(* CODESYS project string-builder.library
   Description: The standard ``CONCAT`` function is really cumbersome to use to build complex
      strings. This library implements a string builder method and some string format
      functions.
   Author: John te Bokkel
   Version: 0.5.0.0
   Company: PowerCore Engineering
   Title: StringBuilder32
   Placeholder: StringBuilder
   LanguageModelAttribute: qualified-access-only
   DefaultNamespace: PSB
   DocFormat: reStructuredText

Project tree, tasks and I/O mapping:
  libraries: CAA Types Extern, 3.5.17.0 (CAA Technical Workgroup); CAA FB Factory, 3.5.17.0 (CAA Technical Workgroup); Common Behaviour Model, 3.5.17.0 (3S - Smart Software Solutions GmbH); StringUtils, 3.5.18.0 (System); StringBuilder Interfaces32, * (PowerCore Engineering); MemoryUtils, * (3S - Smart Software Solutions GmbH)
  StringBuilder/
    Enums/
      data type Alignment
      data type ERROR
    Functions/
      function Align_String [ST]
      function ANY_TO_NUMSTRING [ST]
      function AppendStringNTimes [ST]
      function DIGIT_TO_CHAR [ST]
      FormatExt/
        function FormatExt_10 [ST]
        function FormatExt_1 [ST]
        function FormatExt_2 [ST]
        function FormatExt_3 [ST]
        function FormatExt_4 [ST]
        function FormatExt_5 [ST]
        function FormatExt_6 [ST]
        function FormatExt_7 [ST]
        function FormatExt_8 [ST]
        function FormatExt_9 [ST]
        function FormatExt_ArrayOfStr [ST]
      function Format_10 [ST]
      function Format_1 [ST]
      function Format_2 [ST]
      function Format_3 [ST]
      function Format_4 [ST]
      function Format_5 [ST]
      function Format_6 [ST]
      function Format_7 [ST]
      function Format_8 [ST]
      function Format_9 [ST]
      function Format_ArrayOfStr [ST]
      function POINTER_TO_STRING [ST]
    Function Blocks/
      function block StringBuilderExt [ST]: Append, p_CharBufferPtr, p_length, Reset
      function block StringBuilder [ST]: Append, p_CharBufferPtr, p_length, Reset
    GlobalConstants/
      global variables Constants
    GlobalVariables/
      global variables Variables
    Interfaces/
    Internal/
      function FindFormat [ST]
    Structs/
      data type FormatOptions
      data type slice
    Templates/
      Behaviour Model/
        function block ETrigATlTo_Temp [ST]: CleanupAction, CyclicAction, ExitAction, ResetAction, SampleAction, StartAction
        function block ETrigATl_Temp [ST]: CleanupAction, CyclicAction, ExitAction, ResetAction, SampleAction, StartAction
        function block ETrigATo_Temp [ST]: CleanupAction, CyclicAction, ExitAction, ResetAction, SampleAction, StartAction
        function block ETrigA_Temp [ST]: CleanupAction, CyclicAction, ExitAction, ResetAction, SampleAction, StartAction
        function block ETrigTlTo_Temp [ST]: CleanupAction, CyclicAction, ExitAction, ResetAction, SampleAction, StartAction
        function block ETrigTl_Temp [ST]: CleanupAction, CyclicAction, ExitAction, ResetAction, SampleAction, StartAction
        function block ETrigTo_Temp [ST]: CleanupAction, CyclicAction, ExitAction, ResetAction, SampleAction, StartAction
        function block ETrig_Temp [ST]: CleanupAction, CyclicAction, ExitAction, ResetAction, SampleAction, StartAction
        function block LConC_Temp [ST]: CleanupAction, CyclicAction, ExitAction, ResetAction, StartAction
        function block LConTlC_Temp [ST]: CleanupAction, CyclicAction, ExitAction, ResetAction, StartAction
        function block LConTlTo_Temp [ST]: CleanupAction, CyclicAction, ExitAction, ResetAction, StartAction
        function block LConTl_Temp [ST]: CleanupAction, CyclicAction, ExitAction, ResetAction, StartAction
        function block LConTo_Temp [ST]: CleanupAction, CyclicAction, ExitAction, ResetAction, StartAction
        function block LCon_Temp [ST]: CleanupAction, CyclicAction, ExitAction, ResetAction, StartAction
      FB Factory/
        function block CustomData [ST]
        function block CustomFBFactory_heap [ST]: Create, prvInstCount, prvInstPoolExtendsFactor, prvInstSize
        function block CustomFBFactory_static [ST]: Create, prvInstPoolAdr, prvInstPoolSize, prvInstSize
        function block CustomFB [ST]: prvInstInit
    Types/
*)

// StringBuilder/Enums/Alignment
{attribute 'qualified_only'}
{attribute 'strict'}
TYPE Alignment :
(
	Left,
	Center,
	Right
);
END_TYPE

// StringBuilder/Enums/ERROR
{attribute 'qualified_only'}
//{attribute 'conditionalshow'}
//{attribute 'conditionalshow' := 'SomeText'}
//{attribute 'hide'}
TYPE ERROR : (NO_ERROR, TIME_OUT); END_TYPE

// StringBuilder/Structs/FormatOptions
TYPE FormatOptions :
STRUCT
	// how many decimals a formatted number should have
	iPrecision : INT := -1;
	// the min width of the field in characters (if less than 0 no padding or alignment is performed)
	iMinWidth : INT := -1;
	// how the text is aligned
	align : Alignment := Alignment.Right;
	// A single character which is used to pad the formatted text
	sFill : STRING(1) := ' '; 
END_STRUCT
END_TYPE

// StringBuilder/Structs/slice
TYPE slice :
STRUCT
	start : DINT;
	end : DINT;
END_STRUCT
END_TYPE

// StringBuilder/GlobalConstants/Constants
{attribute 'qualified_only'}
VAR_GLOBAL CONSTANT
	gc_fmtPointerOptions : FormatOptions := (iMinWidth:=16, align:=Alignment.Right, sFill:='0');
END_VAR

// StringBuilder/GlobalVariables/Variables
{attribute 'qualified_only'}
//{attribute 'conditionalshow'}
//{attribute 'conditionalshow' := 'SomeText'}
//{attribute 'hide'}
VAR_GLOBAL
	g_iDummy : INT; /// This is a dummy global variable
END_VAR

// StringBuilder/Functions/Align_String
FUNCTION Align_String : BOOL
VAR_INPUT
	itfStringBuilder : PSBItfs.IStringBuilder;
	sVal : STRING(255);
	options : FormatOptions;
END_VAR
VAR
	iWidth : INT;
	iPadding : INT;
	iLeft : INT;
	iRight : INT;
END_VAR

Align_String := TRUE;
IF itfStringBuilder <> 0 THEN
	IF options.iMinWidth >= 0 THEN
		iWidth := DINT_TO_INT(Stu.StrLenA(ADR(sVal)));
		IF iWidth < options.iMinWidth THEN
			iPadding := options.iMinWidth - iWidth;
		ELSE
			iPadding := 0;
		END_IF
		
		IF iPadding = 0 THEN
			itfStringBuilder.Append(sVal);
			RETURN;
		END_IF
		
		CASE options.align OF
			Alignment.Left:
				itfStringBuilder.Append(sVal);
				AppendStringNTimes(itfStringBuilder, options.sFill, iPadding);
			Alignment.Center:
				iLeft := iPadding / 2;
				iRight := (iPadding + 1) / 2;
				AppendStringNTimes(itfStringBuilder, options.sFill, iLeft);
				itfStringBuilder.Append(sVal);
				AppendStringNTimes(itfStringBuilder, options.sFill, iRight);
			Alignment.Right:
				AppendStringNTimes(itfStringBuilder, options.sFill, iPadding);
				itfStringBuilder.Append(sVal);
		END_CASE
	ELSE
		itfStringBuilder.Append(sVal);
	END_IF
ELSE
	Align_String := FALSE;
END_IF

END_FUNCTION

// StringBuilder/Functions/AppendStringNTimes
FUNCTION AppendStringNTimes : BOOL
VAR_INPUT
	itfStringBuilder : PSBItfs.IStringBuilder;
	sVal : STRING(1);
	iTimes : INT;
END_VAR
VAR
	ix : INT;
END_VAR

AppendStringNTimes := TRUE;
IF itfStringBuilder <> 0 THEN
	IF iTimes > 0 THEN
		FOR ix:=0 TO (iTimes - 1) BY 1 DO
			itfStringBuilder.Append(sVal);
		END_FOR
	END_IF
ELSE
	AppendStringNTimes := FALSE;
END_IF

END_FUNCTION

// StringBuilder/Functions/ANY_TO_NUMSTRING
FUNCTION ANY_TO_NUMSTRING : STRING(129)
VAR_INPUT
	in : ANY;
	base : BYTE;
	xLoCase : BOOL;
	options : FormatOptions;
END_VAR
VAR
	sb : StringBuilder;
	pResult : POINTER TO STRING(129);
	aBuf : ARRAY [0..129] OF BYTE;
	value : UDINT;
	wValue : WORD;
	dwValue : DWORD;
	siValue : SINT;
	iValue : INT;
	diValue : DINT;
	liValue : LINT;
	xSigned : BOOL;
	digit : BYTE;
	ix : BYTE;
	_base : UDINT;
END_VAR

CASE in.TypeClass OF
	__SYSTEM.TYPE_CLASS.TYPE_BOOL:
		value := BYTE_TO_UDINT(in.pValue^);
	__SYSTEM.TYPE_CLASS.TYPE_BIT:
		value := BYTE_TO_UDINT(in.pValue^);
	__SYSTEM.TYPE_CLASS.TYPE_BYTE:
		value := BYTE_TO_UDINT(in.pValue^);
	__SYSTEM.TYPE_CLASS.TYPE_WORD:
		MEMUtils.MemCpy(ADR(wValue), in.pValue, SIZEOF(WORD));
		value := WORD_TO_UDINT(wValue);
	__SYSTEM.TYPE_CLASS.TYPE_DWORD:
		MEMUtils.MemCpy(ADR(dwValue), in.pValue, SIZEOF(DWORD));
		value := DWORD_TO_UDINT(dwValue);
	__SYSTEM.TYPE_CLASS.TYPE_LWORD:
		MEMUtils.MemCpy(ADR(value), in.pValue, SIZEOF(LWORD));
	__SYSTEM.TYPE_CLASS.TYPE_SINT:
		MEMUtils.MemCpy(ADR(siValue), in.pValue, SIZEOF(SINT));
		xSigned := siValue < 0;
		value := SINT_TO_UDINT(ABS(siValue));
	__SYSTEM.TYPE_CLASS.TYPE_INT:
		MEMUtils.MemCpy(ADR(iValue), in.pValue, SIZEOF(INT));
		xSigned := iValue < 0;
		value := INT_TO_UDINT(ABS(iValue));
	__SYSTEM.TYPE_CLASS.TYPE_DINT:
		MEMUtils.MemCpy(ADR(diValue), in.pValue, SIZEOF(DINT));
		xSigned := diValue < 0;
		value := DINT_TO_UDINT(ABS(diValue));
	__SYSTEM.TYPE_CLASS.TYPE_LINT:
		MEMUtils.MemCpy(ADR(liValue), in.pValue, SIZEOF(LINT));
		xSigned := liValue < 0;
		value := LINT_TO_UDINT(ABS(liValue));
	__SYSTEM.TYPE_CLASS.TYPE_USINT:
		value := BYTE_TO_UDINT(in.pValue^);
	__SYSTEM.TYPE_CLASS.TYPE_UINT:
		MEMUtils.MemCpy(ADR(wValue), in.pValue, SIZEOF(UINT));
		value := WORD_TO_UDINT(wValue);
	__SYSTEM.TYPE_CLASS.TYPE_UDINT:
		MEMUtils.MemCpy(ADR(dwValue), in.pValue, SIZEOF(UDINT));
		value := DWORD_TO_UDINT(dwValue);
	__SYSTEM.TYPE_CLASS.TYPE_ULINT:
		MEMUtils.MemCpy(ADR(value), in.pValue, SIZEOF(ULINT));
	__SYSTEM.TYPE_CLASS.TYPE_REAL:
		MEMUtils.MemCpy(ADR(dwValue), in.pValue, SIZEOF(REAL));
		value := DWORD_TO_UDINT(dwValue);
	__SYSTEM.TYPE_CLASS.TYPE_LREAL:
		MEMUtils.MemCpy(ADR(value), in.pValue, SIZEOF(LREAL));
	(* __SYSTEM.TYPE_CLASS.TYPE_STRING:
	__SYSTEM.TYPE_CLASS.TYPE_WSTRING: *)
	__SYSTEM.TYPE_CLASS.TYPE_TIME:
		MEMUtils.MemCpy(ADR(dwValue), in.pValue, SIZEOF(TIME));
		value := DWORD_TO_UDINT(dwValue);
	__SYSTEM.TYPE_CLASS.TYPE_DATE:
		MEMUtils.MemCpy(ADR(dwValue), in.pValue, SIZEOF(DATE));
		value := DWORD_TO_UDINT(dwValue);
	__SYSTEM.TYPE_CLASS.TYPE_DATEANDTIME:
		MEMUtils.MemCpy(ADR(dwValue), in.pValue, SIZEOF(DT));
		value := DWORD_TO_UDINT(dwValue);
	__SYSTEM.TYPE_CLASS.TYPE_TIMEOFDAY:
		MEMUtils.MemCpy(ADR(dwValue), in.pValue, SIZEOF(TOD));
		value := DWORD_TO_UDINT(dwValue);
	(*__SYSTEM.TYPE_CLASS.TYPE_POINTER:
	__SYSTEM.TYPE_CLASS.TYPE_REFERENCE:
	__SYSTEM.TYPE_CLASS.TYPE_SUBRANGE:
	__SYSTEM.TYPE_CLASS.TYPE_ENUM:
	__SYSTEM.TYPE_CLASS.TYPE_ARRAY:
	__SYSTEM.TYPE_CLASS.TYPE_PARAMS:
	__SYSTEM.TYPE_CLASS.TYPE_USERDEF:
	__SYSTEM.TYPE_CLASS.TYPE_NONE:
	__SYSTEM.TYPE_CLASS.TYPE_ANY:
	__SYSTEM.TYPE_CLASS.TYPE_ANYBIT:
	__SYSTEM.TYPE_CLASS.TYPE_ANYDATE:
	__SYSTEM.TYPE_CLASS.TYPE_ANYINT:
	__SYSTEM.TYPE_CLASS.TYPE_ANYNUM:
	__SYSTEM.TYPE_CLASS.TYPE_ANYREAL:
	__SYSTEM.TYPE_CLASS.TYPE_LAZY: *)
	__SYSTEM.TYPE_CLASS.TYPE_LTIME:
		MEMUtils.MemCpy(ADR(value), in.pValue, SIZEOF(LTIME));
	__SYSTEM.TYPE_CLASS.TYPE_LDATE:
		MEMUtils.MemCpy(ADR(value), in.pValue, SIZEOF(LDATE));
	__SYSTEM.TYPE_CLASS.TYPE_LDATEANDTIME:
		MEMUtils.MemCpy(ADR(value), in.pValue, SIZEOF(LDT));
	(*__SYSTEM.TYPE_CLASS.TYPE_BITCONST: *)
	ELSE
		// Anything not explicitly handled will return the pointer value
		value := __XWORD_TO_UDINT(in.pValue);
END_CASE

ix := 129;
_base := BYTE_TO_UDINT(base);
WHILE TRUE DO
	digit := UDINT_TO_BYTE(value MOD _base);
	ix := ix - 1;
	aBuf[ix] := DIGIT_TO_CHAR(digit, xLoCase);
	value := value / _base;
	IF value = 0 OR (xSigned AND ix = 1) OR (NOT xSigned AND ix = 0) THEN
		EXIT;
	END_IF
END_WHILE

IF xSigned THEN
	ix := ix - 1;
	aBuf[ix] := 45; // '-'
END_IF

pResult := ADR(aBuf[ix]);

Align_String(sb, pResult^, options);
ANY_TO_NUMSTRING := sb.sOutput;

END_FUNCTION

// StringBuilder/Functions/DIGIT_TO_CHAR
FUNCTION DIGIT_TO_CHAR : BYTE
VAR_INPUT
	digit : BYTE;
	xLoCase : BOOL;
END_VAR
VAR
END_VAR

IF digit < 10 THEN
	DIGIT_TO_CHAR := digit + 48; // '0' = 48
ELSE
	IF xLoCase THEN
		DIGIT_TO_CHAR := digit + 97 - 10; // 'a' = 97
	ELSE
		DIGIT_TO_CHAR := digit + 65 - 10; // 'A' = 65
	END_IF	
END_IF

END_FUNCTION

// StringBuilder/Function Blocks/StringBuilder
{attribute 'analysis' := '-2'} // empty function block
FUNCTION_BLOCK StringBuilder IMPLEMENTS PSBItfs.IStringBuilder
VAR_INPUT
END_VAR
VAR_OUTPUT
	sOutput : STRING(255);
END_VAR
VAR
	ix : DINT;
END_VAR

METHOD PUBLIC Append : INT
VAR_INPUT
	sVal : STRING(255);
END_VAR
VAR
	diCpy : DINT;
	diCpyInter : DINT;
END_VAR
IF ix = 0 THEN
	sOutput := sVal;
	ix := MAX(Stu.StrLenA(ADR(sOutput)), 0);
	Append := DINT_TO_INT(ix);
ELSIF ix >= 255 THEN
	Append := 0;
ELSE
	
	diCpyInter := Stu.StrCpyA(ADR(sOutput[ix]), MAX(0, 255-ix), ADR(sVal));
	// Working around TM258 PLC StrCpyA not actually returning the number of copied characters
	IF diCpyInter = 0 THEN
		// need to add one for the \0 that StrCpyA should count
		diCpyInter := MIN(Stu.StrLenA(ADR(sVal)) + 1, 255-ix);
	END_IF
	// 1 less than StrCpyA because that value includes \0 (NULL) terminator
	diCpy := MAX(diCpyInter - 1, 0);
	
	Append := DINT_TO_INT(diCpy);
	ix := ix + diCpy;
	// ensure we always have null termination
	sOutput[ix+1] := 0;
END_IF
END_METHOD

PROPERTY p_CharBufferPtr : POINTER TO BYTE
GET
p_CharBufferPtr := ADR(sOutput);
END_GET
END_PROPERTY

PROPERTY p_length : UDINT
GET
p_length := DINT_TO_UDINT(ix);
END_GET
END_PROPERTY

METHOD Reset : BOOL
VAR_INPUT
END_VAR
sOutput := '';
ix := 0;
END_METHOD

END_FUNCTION_BLOCK

// StringBuilder/Functions/Format_10
/// String format ``fmtstr`` with values in ``str1``, etc.
FUNCTION Format_10 : STRING(255)
VAR_INPUT
	fmtstr : STRING(255);
	str1 : STRING(255);
	str2 : STRING(255);
	str3 : STRING(255);
	str4 : STRING(255);
	str5 : STRING(255);
	str6 : STRING(255);
	str7 : STRING(255);
	str8 : STRING(255);
	str9 : STRING(255);
	str10 : STRING(255);
END_VAR
VAR
	apStr : ARRAY [0..9] OF POINTER TO STRING(255) := [ADR(str1), ADR(str2), ADR(str3), ADR(str4), ADR(str5),
	                                                   ADR(str6), ADR(str7), ADR(str8), ADR(str9), ADR(str10)];
END_VAR

Format_10 := Format_ArrayOfStr(fmtstr, ADR(apStr), 10);

END_FUNCTION

// StringBuilder/Functions/Format_ArrayOfStr
/// Replace ``uiElements`` number of ``{}`` with the sequential values in array. 
FUNCTION Format_ArrayOfStr : STRING(255)
VAR_INPUT
	fmtstr : STRING(255);
	// pArray is cast to: POINTER TO ARRAY [0..99] OF POINTER TO STRING(255);
	pArray : POINTER TO BYTE;
	// Actual number of elements in array
	uiElements : UINT;
END_VAR
VAR
	papStr : POINTER TO ARRAY [0..99] OF POINTER TO STRING(255);
	ix : UINT;
	sb : StringBuilder;
	fmtAt : slice;
	last : slice;
	substr : STRING(255);
	iLenRemaining : INT;
	iPos : INT;
END_VAR

papStr := pArray;
fmtAt := FindFormat(fmtstr, 1);

IF fmtAt.start <= 0 THEN
	Format_ArrayOfStr := fmtstr;
	// no format strings found so just return
	RETURN;
END_IF

last.end := 1;
iPos:=1;

FOR ix:=0 TO MIN((uiElements - 1), 99) BY 1 DO
	Stu.StrMidA(pst:=ADR(fmtstr),
				uiInputBufferSize:=SIZEOF(fmtstr),
				iLength:=DINT_TO_INT(fmtAt.start) - iPos,
				iPosition:=iPos,
				pstResult:=ADR(substr),
				uiResultBufferSize:=SIZEOF(substr));
	sb.Append(substr);
	sb.Append(papStr^[ix]^);
	last := fmtAt;
	iPos := DINT_TO_INT(last.end+1);
	fmtAt := FindFormat(fmtstr, fmtAt.end);
	IF fmtAt.start <= 0 THEN
		EXIT;
	END_IF
END_FOR

iLenRemaining := DINT_TO_INT(Stu.StrLenA(ADR(fmtstr[last.end])));
IF iLenRemaining > 0 THEN
	Stu.StrMidA(pst:=ADR(fmtstr),
				uiInputBufferSize:=SIZEOF(fmtstr),
				iLength:=iLenRemaining,
				iPosition:=DINT_TO_INT(last.end+1),
				pstResult:=ADR(substr),
				uiResultBufferSize:=SIZEOF(substr));
	sb.Append(substr);
END_IF
Format_ArrayOfStr := sb.sOutput;

END_FUNCTION

// StringBuilder/Internal/FindFormat
/// Find the format string
{attribute 'conditionalshow' := 'Developer'}
FUNCTION FindFormat : slice
VAR_IN_OUT CONSTANT
	fmtstr : STRING(255);
END_VAR
VAR_INPUT
	start : DINT;
END_VAR
VAR
END_VAR
VAR CONSTANT
	FMT : STRING(2) := '{}';
END_VAR

// lets start out with really basic
// this could evolve into a lexer based system with format directives 
// etc, but lets just start with what we need today.

FindFormat.start := Stu.StrFindA(ADR(fmtstr), ADR(FMT), DINT_TO_UINT(start));
IF FindFormat.start > 0 THEN
	FindFormat.end := FindFormat.start + 1;
END_IF

END_FUNCTION

// StringBuilder/Functions/Format_1
/// String format ``fmtstr`` with values in ``str1``, etc.
FUNCTION Format_1 : STRING(255)
VAR_INPUT
	fmtstr : STRING(255);
	str1 : STRING(255);
END_VAR
VAR
	sb : StringBuilder;
	fmtAt : slice;
	substr : STRING(255);
	iLenRemaining : INT;
END_VAR

fmtAt := FindFormat(fmtstr, 1);
IF fmtAt.start <= 0 THEN
	Format_1 := fmtstr;
ELSE
	Stu.StrMidA(pst:=ADR(fmtstr), uiInputBufferSize:=SIZEOF(fmtstr), iLength:=DINT_TO_INT(fmtAt.start - 1), iPosition:=1, pstResult:=ADR(substr), uiResultBufferSize:=SIZEOF(substr));
	sb.Append(substr);
	sb.Append(str1);
	iLenRemaining := DINT_TO_INT(Stu.StrLenA(ADR(fmtstr[fmtAt.end])));
	IF iLenRemaining > 0 THEN
		Stu.StrMidA(pst:=ADR(fmtstr), uiInputBufferSize:=SIZEOF(fmtstr), iLength:=iLenRemaining, iPosition:=DINT_TO_INT(fmtAt.end+1), pstResult:=ADR(substr), uiResultBufferSize:=SIZEOF(substr));
		sb.Append(substr);
	END_IF
	Format_1 := sb.sOutput;
END_IF

END_FUNCTION

// StringBuilder/Functions/Format_2
/// String format ``fmtstr`` with values in ``str1``, etc.
FUNCTION Format_2 : STRING(255)
VAR_INPUT
	fmtstr : STRING(255);
	str1 : STRING(255);
	str2 : STRING(255);
END_VAR
VAR
	apStr : ARRAY [0..1] OF POINTER TO STRING(255) := [ADR(str1), ADR(str2)];
END_VAR

Format_2 := Format_ArrayOfStr(fmtstr, ADR(apStr), 2);

END_FUNCTION

// StringBuilder/Functions/Format_3
/// String format ``fmtstr`` with values in ``str1``, etc.
FUNCTION Format_3 : STRING(255)
VAR_INPUT
	fmtstr : STRING(255);
	str1 : STRING(255);
	str2 : STRING(255);
	str3 : STRING(255);
END_VAR
VAR
	apStr : ARRAY [0..2] OF POINTER TO STRING(255) := [ADR(str1), ADR(str2), ADR(str3)];
END_VAR

Format_3 := Format_ArrayOfStr(fmtstr, ADR(apStr), 3);

END_FUNCTION

// StringBuilder/Functions/Format_4
/// String format ``fmtstr`` with values in ``str1``, etc.
FUNCTION Format_4 : STRING(255)
VAR_INPUT
	fmtstr : STRING(255);
	str1 : STRING(255);
	str2 : STRING(255);
	str3 : STRING(255);
	str4 : STRING(255);
END_VAR
VAR
	apStr : ARRAY [0..3] OF POINTER TO STRING(255) := [ADR(str1), ADR(str2), ADR(str3), ADR(str4)];
END_VAR

Format_4 := Format_ArrayOfStr(fmtstr, ADR(apStr), 4);

END_FUNCTION

// StringBuilder/Functions/Format_5
/// String format ``fmtstr`` with values in ``str1``, etc.
FUNCTION Format_5 : STRING(255)
VAR_INPUT
	fmtstr : STRING(255);
	str1 : STRING(255);
	str2 : STRING(255);
	str3 : STRING(255);
	str4 : STRING(255);
	str5 : STRING(255);
END_VAR
VAR
	apStr : ARRAY [0..4] OF POINTER TO STRING(255) := [ADR(str1), ADR(str2), ADR(str3), ADR(str4), ADR(str5)];
END_VAR

Format_5 := Format_ArrayOfStr(fmtstr, ADR(apStr), 5);

END_FUNCTION

// StringBuilder/Functions/Format_6
/// String format ``fmtstr`` with values in ``str1``, etc.
FUNCTION Format_6 : STRING(255)
VAR_INPUT
	fmtstr : STRING(255);
	str1 : STRING(255);
	str2 : STRING(255);
	str3 : STRING(255);
	str4 : STRING(255);
	str5 : STRING(255);
	str6 : STRING(255);
END_VAR
VAR
	apStr : ARRAY [0..6] OF POINTER TO STRING(255) := [ADR(str1), ADR(str2), ADR(str3), ADR(str4), ADR(str5),
	                                                   ADR(str6)];
END_VAR

Format_6 := Format_ArrayOfStr(fmtstr, ADR(apStr), 6);

END_FUNCTION

// StringBuilder/Functions/Format_7
/// String format ``fmtstr`` with values in ``str1``, etc.
FUNCTION Format_7 : STRING(255)
VAR_INPUT
	fmtstr : STRING(255);
	str1 : STRING(255);
	str2 : STRING(255);
	str3 : STRING(255);
	str4 : STRING(255);
	str5 : STRING(255);
	str6 : STRING(255);
	str7 : STRING(255);
END_VAR
VAR
	apStr : ARRAY [0..6] OF POINTER TO STRING(255) := [ADR(str1), ADR(str2), ADR(str3), ADR(str4), ADR(str5),
	                                                   ADR(str6), ADR(str7)];
END_VAR

Format_7 := Format_ArrayOfStr(fmtstr, ADR(apStr), 7);

END_FUNCTION

// StringBuilder/Functions/Format_8
/// String format ``fmtstr`` with values in ``str1``, etc.
FUNCTION Format_8 : STRING(255)
VAR_INPUT
	fmtstr : STRING(255);
	str1 : STRING(255);
	str2 : STRING(255);
	str3 : STRING(255);
	str4 : STRING(255);
	str5 : STRING(255);
	str6 : STRING(255);
	str7 : STRING(255);
	str8 : STRING(255);
END_VAR
VAR
	apStr : ARRAY [0..7] OF POINTER TO STRING(255) := [ADR(str1), ADR(str2), ADR(str3), ADR(str4), ADR(str5),
	                                                   ADR(str6), ADR(str7), ADR(str8)];
END_VAR

Format_8 := Format_ArrayOfStr(fmtstr, ADR(apStr), 8);

END_FUNCTION

// StringBuilder/Functions/Format_9
/// String format ``fmtstr`` with values in ``str1``, etc.
FUNCTION Format_9 : STRING(255)
VAR_INPUT
	fmtstr : STRING(255);
	str1 : STRING(255);
	str2 : STRING(255);
	str3 : STRING(255);
	str4 : STRING(255);
	str5 : STRING(255);
	str6 : STRING(255);
	str7 : STRING(255);
	str8 : STRING(255);
	str9 : STRING(255);
END_VAR
VAR
	apStr : ARRAY [0..8] OF POINTER TO STRING(255) := [ADR(str1), ADR(str2), ADR(str3), ADR(str4), ADR(str5),
	                                                   ADR(str6), ADR(str7), ADR(str8), ADR(str9)];
END_VAR

Format_9 := Format_ArrayOfStr(fmtstr, ADR(apStr), 9);

END_FUNCTION

// StringBuilder/Functions/POINTER_TO_STRING
FUNCTION POINTER_TO_STRING : STRING(129)
VAR_INPUT
	ptr : __XWORD;
END_VAR
VAR
	sPtr : STRING(129);
END_VAR

POINTER_TO_STRING := '0x';
sPtr := ANY_TO_NUMSTRING(ptr, 16, TRUE, Constants.gc_fmtPointerOptions);
Stu.StrConcatA(pstFrom:=ADR(sPtr), pstTo:=ADR(POINTER_TO_STRING), SIZEOF(POINTER_TO_STRING));

END_FUNCTION

// StringBuilder/Function Blocks/StringBuilderExt
/// String Builder that takes externally allocated buffer
{attribute 'analysis' := '-2'} // empty function block
FUNCTION_BLOCK StringBuilderExt IMPLEMENTS PSBItfs.IStringBuilder
VAR_INPUT
	pBuffer : POINTER TO BYTE;
	szBuffer : UDINT;
END_VAR
VAR_OUTPUT
END_VAR
VAR
	ix : UDINT;
	psBuffer : POINTER TO STRING(255);
END_VAR

METHOD PUBLIC Append : INT
VAR_INPUT
	sVal : STRING(255);
END_VAR
VAR
	diCpy : DINT;
	diCpyInter : DINT;
	pEnd : POINTER TO BYTE;
	diLen : DINT;
END_VAR
IF pBuffer <> 0 THEN
	psBuffer := pBuffer;
	IF ix = 0 THEN
		psBuffer^ := sVal;
		diLen := MAX(Stu.StrLenA(pBuffer), 0);
		IF diLen > 0 THEN
			ix := DINT_TO_UDINT(diLen);
		END_IF
		Append := UDINT_TO_INT(ix);
	ELSIF ix >= szBuffer THEN
		Append := 0;
	ELSE
		diCpyInter := Stu.StrCpyA(pBuffer + ix, UDINT_TO_DINT(MAX(0, szBuffer-ix)), ADR(sVal));
		// Working around TM258 PLC StrCpyA not actually returning the number of copied characters
		IF diCpyInter = 0 THEN
			// need to add one for the \0 that StrCpyA should count
			diCpyInter := MIN(Stu.StrLenA(ADR(sVal)) + 1, UDINT_TO_DINT(szBuffer - ix));
		END_IF
		// 1 less than StrCpyA because that value includes \0 (NULL) terminator
		diCpy := MAX(diCpyInter - 1, 0);
		
		Append := DINT_TO_INT(diCpy);
		ix := ix + DINT_TO_UDINT(diCpy);
		// ensure we always have null termination
		IF ix < szBuffer THEN
			pEnd := pBuffer + ix + 1;
		ELSE
			pEnd := pBuffer + ix;
		END_IF
		pEnd^ := 0;
	END_IF
ELSE
	Append := -1;
END_IF
END_METHOD

PROPERTY p_CharBufferPtr : POINTER TO BYTE
GET
p_CharBufferPtr := pBuffer;
END_GET
END_PROPERTY

PROPERTY p_length : UDINT
GET
p_length := ix;
END_GET
END_PROPERTY

METHOD Reset : BOOL
VAR_INPUT
END_VAR
IF pBuffer <> 0 THEN
	pBuffer^ := 0;
END_IF
ix := 0;
END_METHOD

END_FUNCTION_BLOCK

// StringBuilder/Functions/FormatExt/FormatExt_10
{attribute 'analysis' := '-22,-19'}
/// String format ``fmtstr`` with values in ``str1``, etc.
FUNCTION FormatExt_10 : POINTER TO BYTE
VAR_INPUT
	sb : PSBItfs.IStringBuilder;
	fmtstr : STRING(255);
	str1 : STRING(255);
	str2 : STRING(255);
	str3 : STRING(255);
	str4 : STRING(255);
	str5 : STRING(255);
	str6 : STRING(255);
	str7 : STRING(255);
	str8 : STRING(255);
	str9 : STRING(255);
	str10 : STRING(255);
END_VAR
VAR
	apStr : ARRAY [0..9] OF POINTER TO STRING(255) := [ADR(str1), ADR(str2), ADR(str3), ADR(str4), ADR(str5),
	                                                   ADR(str6), ADR(str7), ADR(str8), ADR(str9), ADR(str10)];
END_VAR

IF sb <> 0 THEN
	FormatExt_ArrayOfStr(sb, fmtstr, ADR(apStr), 10);
	FormatExt_10 := sb.p_CharBufferPtr;
END_IF

END_FUNCTION

// StringBuilder/Functions/FormatExt/FormatExt_ArrayOfStr
FUNCTION FormatExt_ArrayOfStr : DINT
VAR_INPUT
	// String Builder
	sb : PSBItfs.IStringBuilder;
	// Format String
	fmtstr : STRING(255);
	// pArray is cast to: POINTER TO ARRAY [0..99] OF POINTER TO STRING(255);
	pArray : POINTER TO BYTE;
	// Actual number of elements in array
	uiElements : UINT;
END_VAR
VAR
	papStr : POINTER TO ARRAY [0..99] OF POINTER TO STRING(255);
	ix : UINT;
	fmtAt : slice;
	last : slice;
	substr : STRING(255);
	iLenRemaining : INT;
	iPos : INT;
END_VAR

IF pArray <> 0 AND sb <> 0 THEN
	papStr := pArray;
	fmtAt := FindFormat(fmtstr, 1);
	
	IF fmtAt.start <= 0 THEN
		// no format strings found so just return copy to string builder
		sb.Append(fmtstr);
		FormatExt_ArrayOfStr := UDINT_TO_DINT(sb.p_length);
		RETURN;
	END_IF
	
	last.end := 1;
	iPos:=1;
	
	FOR ix:=0 TO MIN((uiElements - 1), 99) BY 1 DO
		Stu.StrMidA(pst:=ADR(fmtstr),
					uiInputBufferSize:=SIZEOF(fmtstr),
					iLength:=DINT_TO_INT(fmtAt.start) - iPos,
					iPosition:=iPos,
					pstResult:=ADR(substr),
					uiResultBufferSize:=SIZEOF(substr));
		sb.Append(substr);
		sb.Append(papStr^[ix]^);
		last := fmtAt;
		iPos := DINT_TO_INT(last.end+1);
		fmtAt := FindFormat(fmtstr, fmtAt.end);
		IF fmtAt.start <= 0 THEN
			EXIT;
		END_IF
	END_FOR
	
	iLenRemaining := DINT_TO_INT(Stu.StrLenA(ADR(fmtstr[last.end])));
	IF iLenRemaining > INT#0 THEN
		Stu.StrMidA(pst:=ADR(fmtstr),
					uiInputBufferSize:=SIZEOF(fmtstr),
					iLength:=iLenRemaining,
					iPosition:=DINT_TO_INT(last.end+1),
					pstResult:=ADR(substr),
					uiResultBufferSize:=SIZEOF(substr));
		sb.Append(substr);
	END_IF
	FormatExt_ArrayOfStr := UDINT_TO_DINT(sb.p_length);
ELSE
	FormatExt_ArrayOfStr := 0;
END_IF

END_FUNCTION

// StringBuilder/Functions/FormatExt/FormatExt_1
{attribute 'analysis' := '-22,-19'}
/// String format ``fmtstr`` with values in ``str1``, etc.
FUNCTION FormatExt_1 : POINTER TO BYTE
VAR_INPUT
	sb : PSBItfs.IStringBuilder;
	fmtstr : STRING(255);
	str1 : STRING(255);
END_VAR
VAR
	fmtAt : slice;
	substr : STRING(255);
	iLenRemaining : INT;
END_VAR

IF sb <> 0 THEN
	fmtAt := FindFormat(fmtstr, 1);
	IF fmtAt.start <= 0 THEN
		sb.Append(fmtstr);
	ELSE
		Stu.StrMidA(pst:=ADR(fmtstr), uiInputBufferSize:=SIZEOF(fmtstr), iLength:=DINT_TO_INT(fmtAt.start - 1), iPosition:=1, pstResult:=ADR(substr), uiResultBufferSize:=SIZEOF(substr));
		sb.Append(substr);
		sb.Append(str1);
		iLenRemaining := DINT_TO_INT(Stu.StrLenA(ADR(fmtstr[fmtAt.end])));
		IF iLenRemaining > INT#0 THEN
			Stu.StrMidA(pst:=ADR(fmtstr), uiInputBufferSize:=SIZEOF(fmtstr), iLength:=iLenRemaining, iPosition:=DINT_TO_INT(fmtAt.end+1), pstResult:=ADR(substr), uiResultBufferSize:=SIZEOF(substr));
			sb.Append(substr);
		END_IF
		FormatExt_1 := sb.p_CharBufferPtr;
	END_IF
END_IF

END_FUNCTION

// StringBuilder/Functions/FormatExt/FormatExt_2
{attribute 'analysis' := '-22,-19'}
/// String format ``fmtstr`` with values in ``str1``, etc.
FUNCTION FormatExt_2 : POINTER TO BYTE
VAR_INPUT
	sb : PSBItfs.IStringBuilder;
	fmtstr : STRING(255);
	str1 : STRING(255);
	str2 : STRING(255);
END_VAR
VAR
	apStr : ARRAY [0..1] OF POINTER TO STRING(255) := [ADR(str1), ADR(str2)];
END_VAR

IF sb <> 0 THEN
	FormatExt_ArrayOfStr(sb, fmtstr, ADR(apStr), 2);
	FormatExt_2 := sb.p_CharBufferPtr;
END_IF

END_FUNCTION

// StringBuilder/Functions/FormatExt/FormatExt_3
{attribute 'analysis' := '-22,-19'}
/// String format ``fmtstr`` with values in ``str1``, etc.
FUNCTION FormatExt_3 : POINTER TO BYTE
VAR_INPUT
	sb : PSBItfs.IStringBuilder;
	fmtstr : STRING(255);
	str1 : STRING(255);
	str2 : STRING(255);
	str3 : STRING(255);
END_VAR
VAR
	apStr : ARRAY [0..2] OF POINTER TO STRING(255) := [ADR(str1), ADR(str2), ADR(str3)];
END_VAR

IF sb <> 0 THEN
	FormatExt_ArrayOfStr(sb, fmtstr, ADR(apStr), 3);
	FormatExt_3 := sb.p_CharBufferPtr;
END_IF

END_FUNCTION

// StringBuilder/Functions/FormatExt/FormatExt_4
{attribute 'analysis' := '-22,-19'}
/// String format ``fmtstr`` with values in ``str1``, etc.
FUNCTION FormatExt_4 : POINTER TO BYTE
VAR_INPUT
	sb : PSBItfs.IStringBuilder;
	fmtstr : STRING(255);
	str1 : STRING(255);
	str2 : STRING(255);
	str3 : STRING(255);
	str4 : STRING(255);
END_VAR
VAR
	apStr : ARRAY [0..3] OF POINTER TO STRING(255) := [ADR(str1), ADR(str2), ADR(str3), ADR(str4)];
END_VAR

IF sb <> 0 THEN
	FormatExt_ArrayOfStr(sb, fmtstr, ADR(apStr), 4);
	FormatExt_4 := sb.p_CharBufferPtr;
END_IF

END_FUNCTION

// StringBuilder/Functions/FormatExt/FormatExt_5
{attribute 'analysis' := '-22,-19'}
/// String format ``fmtstr`` with values in ``str1``, etc.
FUNCTION FormatExt_5 : POINTER TO BYTE
VAR_INPUT
	sb : PSBItfs.IStringBuilder;
	fmtstr : STRING(255);
	str1 : STRING(255);
	str2 : STRING(255);
	str3 : STRING(255);
	str4 : STRING(255);
	str5 : STRING(255);
END_VAR
VAR
	apStr : ARRAY [0..4] OF POINTER TO STRING(255) := [ADR(str1), ADR(str2), ADR(str3), ADR(str4), ADR(str5)];
END_VAR

IF sb <> 0 THEN
	FormatExt_ArrayOfStr(sb, fmtstr, ADR(apStr), 5);
	FormatExt_5 := sb.p_CharBufferPtr;
END_IF

END_FUNCTION

// StringBuilder/Functions/FormatExt/FormatExt_6
{attribute 'analysis' := '-22,-19'}
/// String format ``fmtstr`` with values in ``str1``, etc.
FUNCTION FormatExt_6 : POINTER TO BYTE
VAR_INPUT
	sb : PSBItfs.IStringBuilder;
	fmtstr : STRING(255);
	str1 : STRING(255);
	str2 : STRING(255);
	str3 : STRING(255);
	str4 : STRING(255);
	str5 : STRING(255);
	str6 : STRING(255);
END_VAR
VAR
	apStr : ARRAY [0..5] OF POINTER TO STRING(255) := [ADR(str1), ADR(str2), ADR(str3), ADR(str4), ADR(str5),
	                                                   ADR(str6)];
END_VAR

IF sb <> 0 THEN
	FormatExt_ArrayOfStr(sb, fmtstr, ADR(apStr), 6);
	FormatExt_6 := sb.p_CharBufferPtr;
END_IF

END_FUNCTION

// StringBuilder/Functions/FormatExt/FormatExt_7
{attribute 'analysis' := '-22,-19'}
/// String format ``fmtstr`` with values in ``str1``, etc.
FUNCTION FormatExt_7 : POINTER TO BYTE
VAR_INPUT
	sb : PSBItfs.IStringBuilder;
	fmtstr : STRING(255);
	str1 : STRING(255);
	str2 : STRING(255);
	str3 : STRING(255);
	str4 : STRING(255);
	str5 : STRING(255);
	str6 : STRING(255);
	str7 : STRING(255);
END_VAR
VAR
	apStr : ARRAY [0..6] OF POINTER TO STRING(255) := [ADR(str1), ADR(str2), ADR(str3), ADR(str4), ADR(str5),
	                                                   ADR(str6), ADR(str7)];
END_VAR

IF sb <> 0 THEN
	FormatExt_ArrayOfStr(sb, fmtstr, ADR(apStr), 7);
	FormatExt_7 := sb.p_CharBufferPtr;
END_IF

END_FUNCTION

// StringBuilder/Functions/FormatExt/FormatExt_8
{attribute 'analysis' := '-22,-19'}
/// String format ``fmtstr`` with values in ``str1``, etc.
FUNCTION FormatExt_8 : POINTER TO BYTE
VAR_INPUT
	sb : PSBItfs.IStringBuilder;
	fmtstr : STRING(255);
	str1 : STRING(255);
	str2 : STRING(255);
	str3 : STRING(255);
	str4 : STRING(255);
	str5 : STRING(255);
	str6 : STRING(255);
	str7 : STRING(255);
	str8 : STRING(255);
END_VAR
VAR
	apStr : ARRAY [0..7] OF POINTER TO STRING(255) := [ADR(str1), ADR(str2), ADR(str3), ADR(str4), ADR(str5),
	                                                   ADR(str6), ADR(str7), ADR(str8)];
END_VAR

IF sb <> 0 THEN
	FormatExt_ArrayOfStr(sb, fmtstr, ADR(apStr), 8);
	FormatExt_8 := sb.p_CharBufferPtr;
END_IF

END_FUNCTION

// StringBuilder/Functions/FormatExt/FormatExt_9
{attribute 'analysis' := '-22,-19'}
/// String format ``fmtstr`` with values in ``str1``, etc.
FUNCTION FormatExt_9 : POINTER TO BYTE
VAR_INPUT
	sb : PSBItfs.IStringBuilder;
	fmtstr : STRING(255);
	str1 : STRING(255);
	str2 : STRING(255);
	str3 : STRING(255);
	str4 : STRING(255);
	str5 : STRING(255);
	str6 : STRING(255);
	str7 : STRING(255);
	str8 : STRING(255);
	str9 : STRING(255);
END_VAR
VAR
	apStr : ARRAY [0..8] OF POINTER TO STRING(255) := [ADR(str1), ADR(str2), ADR(str3), ADR(str4), ADR(str5),
	                                                   ADR(str6), ADR(str7), ADR(str8), ADR(str9)];
END_VAR

IF sb <> 0 THEN
	FormatExt_ArrayOfStr(sb, fmtstr, ADR(apStr), 9);
	FormatExt_9 := sb.p_CharBufferPtr;
END_IF

END_FUNCTION

// StringBuilder/Templates/Behaviour Model/ETrigATlTo_Temp
//{attribute 'hide_all_locals'}
//{attribute 'conditionalshow_all_locals' := 'SomeText'}
//{attribute 'conditionalshow_all_locals'}
//{attribute 'conditionalshow' := 'SomeText'}
//{attribute 'conditionalshow'}
//{attribute 'hide'}
FUNCTION_BLOCK ETrigATlTo_Temp EXTENDS CBML.ETrigATlTo
VAR_INPUT
	(* specific Inputs *)
END_VAR
VAR_OUTPUT
	(* specific Outputs *)
	eErrorID : ERROR;
END_VAR
VAR
	(* specific vars *)
END_VAR

SUPER^();
IF _Model.iErrorID = CBML.ERROR.TIME_OUT THEN
	eErrorID := ERROR.TIME_OUT;
ELSE
	eErrorID := _Model.iErrorID;
END_IF

METHOD CleanupAction
VAR_INPUT
    xAbortProposed : BOOL;
    iErrorIDProposed: INT;
END_VAR
VAR_OUTPUT
    xComplete : BOOL := TRUE;
    xAbort: BOOL := xAbortProposed;
 	iErrorID : INT := iErrorIDProposed;
END_VAR
{analysis -2} 
/// ``CleanupAction`` is running until one of the following events occurs:
/// When ``xComplete`` is ``TRUE`` the state |STATE.DONE| is reached.
/// When ``xAbort`` is ``TRUE`` the state |STATE.ABORTED| is reached.
/// When ``iErrorID`` ≠ 0 (Zero) the state |STATE.ERROR| is reached.
///
/// | After a *Ready Condition* as input (``iErrorIDProposed`` = 0 and ``xAbortProposed`` = ``FALSE``), only the output states
/// | `DONE` (``xComplete`` is ``TRUE``) or `ERROR` (``iErrorID`` ≠ 0) are possible.
///
/// | After a *Error Condition* as input (``iErrorIDProposed`` ≠ 0), only the output state
/// | `ERROR` (``iErrorID`` ≠ 0) is possible.
///
/// | After a *Abort Condition* as Input (``xAbortProposed`` = ``TRUE``), only the output states
/// | `ABORTED` (``xAbort`` is ``TRUE``) or `ERROR` (``iErrorID`` ≠ 0) are possible.
///
/// .. admonition:: Example
///
///     .. code-block:: codesys
///     
///         (* common cleanup -- first steps *) 
///         
///         IF xComplete THEN
///             IF xAbortProposed THEN
///                 (* abort condition -- abort specific cleanup *)
///                 xAbort := TRUE;
///                 xComplete := FALSE;
///             ELSIF iErrorIDProposed <> 0 THEN
///                 (* error condition -- error specific cleanup *)
///                 iErrorID := SEL(xComplete, 0, iErrorIDProposed);
///                 xComplete := FALSE;
///             ELSE
///                 (* ready condition -- done specific cleanup*)
///             END_IF
///         END_IF
///
///         (* common cleanup -- last steps *) 
///
/// .. note::
///
///    If this method will not provide any implementation, please remove it!
END_METHOD

METHOD CyclicAction
VAR_INPUT
    itfTimingController : CBML.ITimingController;
END_VAR
VAR_OUTPUT
    xComplete : BOOL := TRUE;
    iErrorID : INT := 0;
END_VAR
{analysis -2} 
/// The CyclicAction is running until either ``xComplete`` is ``TRUE`` or ``iErrorID`` ≠  0 (Zero).
/// If ``xComplete`` is ``TRUE`` or ``iErrorID`` ≠  0 (Zero) the state |STATE.CLEANING| is reached.
/// With ``itfTimingController`` ≠  0 (Zero) it is possible to check the current invocation time (see: |ITimingController.ControllerCheckTiming|).
/// Function blocks with a ``udiTimeLimit`` input variable (see: |IETrigTl|, |IETrigATl|, |IETrigTlTo|, |IETrigATlTo|, |ILConTl|, |ILConTlTo|, |ILConTlC|)
/// should be implement in such a way that the current invocation is exited when the consumed time for this invocation has exceeded the settings from udiTimeLimit.
///
/// .. admonition:: Example
///
///     .. code-block:: codesys
///     
///         REPEAT
///             // working to reach the ready condition
///             // ⇒ xComplete := TRUE
///             // if the maximum invocation time is reached
///             // ⇒ xTimeLimit := TRUE
///             // if the maximum operating time is reached
///             // ⇒ xTimeOut := TRUE
///             // if an error condition is reached
///             // ⇒ set iErrorID to a value other than 0 (Zero)
///             itfTimingController.ControllerCheckTiming(
///                 xTimeOut=>xTimeOut,
///                 xTimeLimit=>xTimeLimit
///             );
///         
///             xComplete := TRUE;
///             iErrorID := ERROR.NO_ERROR;
///     
///         UNTIL xComplete OR
///               xTimeOut OR xTimeLimit OR
///               iErrorID <> ERROR.NO_ERROR
///         END_REPEAT
///
/// .. note::
///
///    If this method will not provide any implementation, please remove it!
END_METHOD

METHOD ExitAction
VAR_INPUT
    xAfterCleanup : BOOL;
    xInCopyCode : BOOL;
END_VAR
{analysis -2} 
/// This method is intended for releasing external resources (like RTS handles).
/// Do not call other internal function block instances in the context of this method.
/// Call only external functions defined inside the RTS.
/// For cleaning up other resources then external ones, please use the ``CleanupAction``.
/// This method should be callable in the context of ``FB_EXIT`` for example
/// before downloading a new application or before reseting an application.
///
/// .. note::
///
///    If this method will not provide any implementation, please remove it!
END_METHOD

METHOD ResetAction
VAR_OUTPUT
    xComplete : BOOL := TRUE;
END_VAR
{analysis -2} 
/// The ``ResetAction`` is running until the output ``xComplete`` is ``TRUE``.
/// If ``xComplete`` is ``TRUE`` the state |STATE.DORMANT| is reached.
///
/// .. note::
///
///    If this method will not provide any implementation, please remove it!
END_METHOD

METHOD SampleAction
VAR_OUTPUT
 	iErrorID : INT := 0;
END_VAR
{analysis -2} 
/// After leaving the state |STATE.DORMANT| the ``SampleAction`` is running one time then the state |STATE.STARTING| is reached.
/// If there is a ``iErrorID`` ≠  0 (Zero) the state |STATE.CLEANING| is reached instead.
///
/// .. note::
///
///    If this method will not provide any implementation, please remove it!
END_METHOD

METHOD StartAction
VAR_OUTPUT
    xComplete : BOOL := TRUE;
	iErrorID : INT := 0;
END_VAR
{analysis -2} 
/// The ``StartAction`` is running until either the output ``xComplete`` is ``TRUE`` or ``iErrorID`` ≠ 0 (Zero).
/// If ``xComplete`` is ``TRUE`` the state |STATE.EXECUTING| is reached.
/// If there is a ``iErrorID`` ≠  0 (Zero) the state |STATE.CLEANING| is reached.
///
/// .. note::
///
///    To sample the inputs in the first invocation of a function block the method SampleAction is the solution of choice.
///    See: |ISampleActionProvider.SampleAction|
///
/// .. note::
///
///    If this method will not provide any implementation, please remove it!
END_METHOD

END_FUNCTION_BLOCK

// StringBuilder/Templates/Behaviour Model/ETrigATl_Temp
//{attribute 'hide_all_locals'}
//{attribute 'conditionalshow_all_locals' := 'SomeText'}
//{attribute 'conditionalshow_all_locals'}
//{attribute 'conditionalshow' := 'SomeText'}
//{attribute 'conditionalshow'}
//{attribute 'hide'}
FUNCTION_BLOCK ETrigATl_Temp EXTENDS CBML.ETrigATl
VAR_INPUT
	(* specific Inputs *)
END_VAR
VAR_OUTPUT
	eErrorID : ERROR;
	(* specific Outputs *)
END_VAR
VAR
	(* specific vars *)
END_VAR

SUPER^();
eErrorID := _Model.iErrorID;

METHOD CleanupAction
VAR_INPUT
    xAbortProposed : BOOL;
    iErrorIDProposed: INT;
END_VAR
VAR_OUTPUT
    xComplete : BOOL := TRUE;
    xAbort: BOOL := xAbortProposed;
 	iErrorID : INT := iErrorIDProposed;
END_VAR
{analysis -2} 
/// ``CleanupAction`` is running until one of the following events occurs:
/// When ``xComplete`` is ``TRUE`` the state |STATE.DONE| is reached.
/// When ``xAbort`` is ``TRUE`` the state |STATE.ABORTED| is reached.
/// When ``iErrorID`` ≠ 0 (Zero) the state |STATE.ERROR| is reached.
///
/// | After a *Ready Condition* as input (``iErrorIDProposed`` = 0 and ``xAbortProposed`` = ``FALSE``), only the output states
/// | `DONE` (``xComplete`` is ``TRUE``) or `ERROR` (``iErrorID`` ≠ 0) are possible.
///
/// | After a *Error Condition* as input (``iErrorIDProposed`` ≠ 0), only the output state
/// | `ERROR` (``iErrorID`` ≠ 0) is possible.
///
/// | After a *Abort Condition* as Input (``xAbortProposed`` = ``TRUE``), only the output states
/// | `ABORTED` (``xAbort`` is ``TRUE``) or `ERROR` (``iErrorID`` ≠ 0) are possible.
///
/// .. admonition:: Example
///
///     .. code-block:: codesys
///     
///         (* common cleanup -- first steps *) 
///         
///         IF xComplete THEN
///             IF xAbortProposed THEN
///                 (* abort condition -- abort specific cleanup *)
///                 xAbort := TRUE;
///                 xComplete := FALSE;
///             ELSIF iErrorIDProposed <> 0 THEN
///                 (* error condition -- error specific cleanup *)
///                 iErrorID := SEL(xComplete, 0, iErrorIDProposed);
///                 xComplete := FALSE;
///             ELSE
///                 (* ready condition -- done specific cleanup*)
///             END_IF
///         END_IF
///
///         (* common cleanup -- last steps *) 
///
/// .. note::
///
///    If this method will not provide any implementation, please remove it!
END_METHOD

METHOD CyclicAction
VAR_INPUT
    itfTimingController : CBML.ITimingController;
END_VAR
VAR_OUTPUT
    xComplete : BOOL := TRUE;
    iErrorID : INT := 0;
END_VAR
{analysis -2} 
/// The CyclicAction is running until either ``xComplete`` is ``TRUE`` or ``iErrorID`` ≠  0 (Zero).
/// If ``xComplete`` is ``TRUE`` or ``iErrorID`` ≠  0 (Zero) the state |STATE.CLEANING| is reached.
/// With ``itfTimingController`` ≠  0 (Zero) it is possible to check the current invocation time (see: |ITimingController.ControllerCheckTiming|).
/// Function blocks with a ``udiTimeLimit`` input variable (see: |IETrigTl|, |IETrigATl|, |IETrigTlTo|, |IETrigATlTo|, |ILConTl|, |ILConTlTo|, |ILConTlC|)
/// should be implement in such a way that the current invocation is exited when the consumed time for this invocation has exceeded the settings from udiTimeLimit.
///
/// .. admonition:: Example
///
///     .. code-block:: codesys
///     
///         REPEAT
///             // working to reach the ready condition
///             // ⇒ xComplete := TRUE
///             // if the maximum invocation time is reached
///             // ⇒ xTimeLimit := TRUE
///             // if the maximum operating time is reached
///             // ⇒ xTimeOut := TRUE
///             // if an error condition is reached
///             // ⇒ set iErrorID to a value other than 0 (Zero)
///             itfTimingController.ControllerCheckTiming(
///                 xTimeOut=>xTimeOut,
///                 xTimeLimit=>xTimeLimit
///             );
///         
///             xComplete := TRUE;
///             iErrorID := ERROR.NO_ERROR;
///     
///         UNTIL xComplete OR
///               xTimeOut OR xTimeLimit OR
///               iErrorID <> ERROR.NO_ERROR
///         END_REPEAT
///
/// .. note::
///
///    If this method will not provide any implementation, please remove it!
END_METHOD

METHOD ExitAction
VAR_INPUT
    xAfterCleanup : BOOL;
    xInCopyCode : BOOL;
END_VAR
{analysis -2} 
/// This method is intended for releasing external resources (like RTS handles).
/// Do not call other internal function block instances in the context of this method.
/// Call only external functions defined inside the RTS.
/// For cleaning up other resources then external ones, please use the ``CleanupAction``.
/// This method should be callable in the context of ``FB_EXIT`` for example
/// before downloading a new application or before reseting an application.
///
/// .. note::
///
///    If this method will not provide any implementation, please remove it!
END_METHOD

METHOD ResetAction
VAR_OUTPUT
    xComplete : BOOL := TRUE;
END_VAR
{analysis -2} 
/// The ``ResetAction`` is running until the output ``xComplete`` is ``TRUE``.
/// If ``xComplete`` is ``TRUE`` the state |STATE.DORMANT| is reached.
///
/// .. note::
///
///    If this method will not provide any implementation, please remove it!
END_METHOD

METHOD SampleAction
VAR_OUTPUT
 	iErrorID : INT := 0;
END_VAR
{analysis -2} 
/// After leaving the state |STATE.DORMANT| the ``SampleAction`` is running one time then the state |STATE.STARTING| is reached.
/// If there is a ``iErrorID`` ≠  0 (Zero) the state |STATE.CLEANING| is reached instead.
///
/// .. note::
///
///    If this method will not provide any implementation, please remove it!
END_METHOD

METHOD StartAction
VAR_OUTPUT
    xComplete : BOOL := TRUE;
	iErrorID : INT := 0;
END_VAR
{analysis -2} 
/// The ``StartAction`` is running until either the output ``xComplete`` is ``TRUE`` or ``iErrorID`` ≠ 0 (Zero).
/// If ``xComplete`` is ``TRUE`` the state |STATE.EXECUTING| is reached.
/// If there is a ``iErrorID`` ≠  0 (Zero) the state |STATE.CLEANING| is reached.
///
/// .. note::
///
///    To sample the inputs in the first invocation of a function block the method SampleAction is the solution of choice.
///    See: |ISampleActionProvider.SampleAction|
///
/// .. note::
///
///    If this method will not provide any implementation, please remove it!
END_METHOD

END_FUNCTION_BLOCK

// StringBuilder/Templates/Behaviour Model/ETrigATo_Temp
//{attribute 'hide_all_locals'}
//{attribute 'conditionalshow_all_locals' := 'SomeText'}
//{attribute 'conditionalshow_all_locals'}
//{attribute 'conditionalshow' := 'SomeText'}
//{attribute 'conditionalshow'}
//{attribute 'hide'}
FUNCTION_BLOCK ETrigATo_Temp EXTENDS CBML.ETrigATo
VAR_INPUT
	(* specific Inputs *)
END_VAR
VAR_OUTPUT
	eErrorID : ERROR;
	(* specific Outputs *)
END_VAR
VAR
	(* specific vars *)
END_VAR

SUPER^();
IF _Model.iErrorID = CBML.ERROR.TIME_OUT THEN
	eErrorID := ERROR.TIME_OUT;
ELSE
	eErrorID := _Model.iErrorID;
END_IF

METHOD CleanupAction
VAR_INPUT
    xAbortProposed : BOOL;
    iErrorIDProposed: INT;
END_VAR
VAR_OUTPUT
    xComplete : BOOL := TRUE;
    xAbort: BOOL := xAbortProposed;
 	iErrorID : INT := iErrorIDProposed;
END_VAR
{analysis -2} 
/// ``CleanupAction`` is running until one of the following events occurs:
/// When ``xComplete`` is ``TRUE`` the state |STATE.DONE| is reached.
/// When ``xAbort`` is ``TRUE`` the state |STATE.ABORTED| is reached.
/// When ``iErrorID`` ≠ 0 (Zero) the state |STATE.ERROR| is reached.
///
/// | After a *Ready Condition* as input (``iErrorIDProposed`` = 0 and ``xAbortProposed`` = ``FALSE``), only the output states
/// | `DONE` (``xComplete`` is ``TRUE``) or `ERROR` (``iErrorID`` ≠ 0) are possible.
///
/// | After a *Error Condition* as input (``iErrorIDProposed`` ≠ 0), only the output state
/// | `ERROR` (``iErrorID`` ≠ 0) is possible.
///
/// | After a *Abort Condition* as Input (``xAbortProposed`` = ``TRUE``), only the output states
/// | `ABORTED` (``xAbort`` is ``TRUE``) or `ERROR` (``iErrorID`` ≠ 0) are possible.
///
/// .. admonition:: Example
///
///     .. code-block:: codesys
///     
///         (* common cleanup -- first steps *) 
///         
///         IF xComplete THEN
///             IF xAbortProposed THEN
///                 (* abort condition -- abort specific cleanup *)
///                 xAbort := TRUE;
///                 xComplete := FALSE;
///             ELSIF iErrorIDProposed <> 0 THEN
///                 (* error condition -- error specific cleanup *)
///                 iErrorID := SEL(xComplete, 0, iErrorIDProposed);
///                 xComplete := FALSE;
///             ELSE
///                 (* ready condition -- done specific cleanup*)
///             END_IF
///         END_IF
///
///         (* common cleanup -- last steps *) 
///
/// .. note::
///
///    If this method will not provide any implementation, please remove it!
END_METHOD

METHOD CyclicAction
VAR_INPUT
    itfTimingController : CBML.ITimingController;
END_VAR
VAR_OUTPUT
    xComplete : BOOL := TRUE;
    iErrorID : INT := 0;
END_VAR
{analysis -2} 
/// The CyclicAction is running until either ``xComplete`` is ``TRUE`` or ``iErrorID`` ≠  0 (Zero).
/// If ``xComplete`` is ``TRUE`` or ``iErrorID`` ≠  0 (Zero) the state |STATE.CLEANING| is reached.
/// With ``itfTimingController`` ≠  0 (Zero) it is possible to check the current invocation time (see: |ITimingController.ControllerCheckTiming|).
/// Function blocks with a ``udiTimeLimit`` input variable (see: |IETrigTl|, |IETrigATl|, |IETrigTlTo|, |IETrigATlTo|, |ILConTl|, |ILConTlTo|, |ILConTlC|)
/// should be implement in such a way that the current invocation is exited when the consumed time for this invocation has exceeded the settings from udiTimeLimit.
///
/// .. admonition:: Example
///
///     .. code-block:: codesys
///     
///         REPEAT
///             // working to reach the ready condition
///             // ⇒ xComplete := TRUE
///             // if the maximum invocation time is reached
///             // ⇒ xTimeLimit := TRUE
///             // if the maximum operating time is reached
///             // ⇒ xTimeOut := TRUE
///             // if an error condition is reached
///             // ⇒ set iErrorID to a value other than 0 (Zero)
///             itfTimingController.ControllerCheckTiming(
///                 xTimeOut=>xTimeOut,
///                 xTimeLimit=>xTimeLimit
///             );
///         
///             xComplete := TRUE;
///             iErrorID := ERROR.NO_ERROR;
///     
///         UNTIL xComplete OR
///               xTimeOut OR xTimeLimit OR
///               iErrorID <> ERROR.NO_ERROR
///         END_REPEAT
///
/// .. note::
///
///    If this method will not provide any implementation, please remove it!
END_METHOD

METHOD ExitAction
VAR_INPUT
    xAfterCleanup : BOOL;
    xInCopyCode : BOOL;
END_VAR
{analysis -2} 
/// This method is intended for releasing external resources (like RTS handles).
/// Do not call other internal function block instances in the context of this method.
/// Call only external functions defined inside the RTS.
/// For cleaning up other resources then external ones, please use the ``CleanupAction``.
/// This method should be callable in the context of ``FB_EXIT`` for example
/// before downloading a new application or before reseting an application.
///
/// .. note::
///
///    If this method will not provide any implementation, please remove it!
END_METHOD

METHOD ResetAction
VAR_OUTPUT
    xComplete : BOOL := TRUE;
END_VAR
{analysis -2} 
/// The ``ResetAction`` is running until the output ``xComplete`` is ``TRUE``.
/// If ``xComplete`` is ``TRUE`` the state |STATE.DORMANT| is reached.
///
/// .. note::
///
///    If this method will not provide any implementation, please remove it!
END_METHOD

METHOD SampleAction
VAR_OUTPUT
 	iErrorID : INT := 0;
END_VAR
{analysis -2} 
/// After leaving the state |STATE.DORMANT| the ``SampleAction`` is running one time then the state |STATE.STARTING| is reached.
/// If there is a ``iErrorID`` ≠  0 (Zero) the state |STATE.CLEANING| is reached instead.
///
/// .. note::
///
///    If this method will not provide any implementation, please remove it!
END_METHOD

METHOD StartAction
VAR_OUTPUT
    xComplete : BOOL := TRUE;
	iErrorID : INT := 0;
END_VAR
{analysis -2} 
/// The ``StartAction`` is running until either the output ``xComplete`` is ``TRUE`` or ``iErrorID`` ≠ 0 (Zero).
/// If ``xComplete`` is ``TRUE`` the state |STATE.EXECUTING| is reached.
/// If there is a ``iErrorID`` ≠  0 (Zero) the state |STATE.CLEANING| is reached.
///
/// .. note::
///
///    To sample the inputs in the first invocation of a function block the method SampleAction is the solution of choice.
///    See: |ISampleActionProvider.SampleAction|
///
/// .. note::
///
///    If this method will not provide any implementation, please remove it!
END_METHOD

END_FUNCTION_BLOCK

// StringBuilder/Templates/Behaviour Model/ETrigA_Temp
//{attribute 'hide_all_locals'}
//{attribute 'conditionalshow_all_locals' := 'SomeText'}
//{attribute 'conditionalshow_all_locals'}
//{attribute 'conditionalshow' := 'SomeText'}
//{attribute 'conditionalshow'}
//{attribute 'hide'}
FUNCTION_BLOCK ETrigA_Temp EXTENDS CBML.ETrigA
VAR_INPUT
	(* specific Inputs *)
END_VAR
VAR_OUTPUT
	eErrorID : ERROR;
	(* specific Outputs *)
END_VAR
VAR
	(* specific vars *)
END_VAR

SUPER^();
eErrorID := _Model.iErrorID;

METHOD CleanupAction
VAR_INPUT
    xAbortProposed : BOOL;
    iErrorIDProposed: INT;
END_VAR
VAR_OUTPUT
    xComplete : BOOL := TRUE;
    xAbort: BOOL := xAbortProposed;
 	iErrorID : INT := iErrorIDProposed;
END_VAR
{analysis -2} 
/// ``CleanupAction`` is running until one of the following events occurs:
/// When ``xComplete`` is ``TRUE`` the state |STATE.DONE| is reached.
/// When ``xAbort`` is ``TRUE`` the state |STATE.ABORTED| is reached.
/// When ``iErrorID`` ≠ 0 (Zero) the state |STATE.ERROR| is reached.
///
/// | After a *Ready Condition* as input (``iErrorIDProposed`` = 0 and ``xAbortProposed`` = ``FALSE``), only the output states
/// | `DONE` (``xComplete`` is ``TRUE``) or `ERROR` (``iErrorID`` ≠ 0) are possible.
///
/// | After a *Error Condition* as input (``iErrorIDProposed`` ≠ 0), only the output state
/// | `ERROR` (``iErrorID`` ≠ 0) is possible.
///
/// | After a *Abort Condition* as Input (``xAbortProposed`` = ``TRUE``), only the output states
/// | `ABORTED` (``xAbort`` is ``TRUE``) or `ERROR` (``iErrorID`` ≠ 0) are possible.
///
/// .. admonition:: Example
///
///     .. code-block:: codesys
///     
///         (* common cleanup -- first steps *) 
///         
///         IF xComplete THEN
///             IF xAbortProposed THEN
///                 (* abort condition -- abort specific cleanup *)
///                 xAbort := TRUE;
///                 xComplete := FALSE;
///             ELSIF iErrorIDProposed <> 0 THEN
///                 (* error condition -- error specific cleanup *)
///                 iErrorID := SEL(xComplete, 0, iErrorIDProposed);
///                 xComplete := FALSE;
///             ELSE
///                 (* ready condition -- done specific cleanup*)
///             END_IF
///         END_IF
///
///         (* common cleanup -- last steps *) 
///
/// .. note::
///
///    If this method will not provide any implementation, please remove it!
END_METHOD

METHOD CyclicAction
VAR_INPUT
    itfTimingController : CBML.ITimingController;
END_VAR
VAR_OUTPUT
    xComplete : BOOL := TRUE;
    iErrorID : INT := 0;
END_VAR
{analysis -2} 
/// The CyclicAction is running until either ``xComplete`` is ``TRUE`` or ``iErrorID`` ≠  0 (Zero).
/// If ``xComplete`` is ``TRUE`` or ``iErrorID`` ≠  0 (Zero) the state |STATE.CLEANING| is reached.
/// With ``itfTimingController`` ≠  0 (Zero) it is possible to check the current invocation time (see: |ITimingController.ControllerCheckTiming|).
/// Function blocks with a ``udiTimeLimit`` input variable (see: |IETrigTl|, |IETrigATl|, |IETrigTlTo|, |IETrigATlTo|, |ILConTl|, |ILConTlTo|, |ILConTlC|)
/// should be implement in such a way that the current invocation is exited when the consumed time for this invocation has exceeded the settings from udiTimeLimit.
///
/// .. admonition:: Example
///
///     .. code-block:: codesys
///     
///         REPEAT
///             // working to reach the ready condition
///             // ⇒ xComplete := TRUE
///             // if the maximum invocation time is reached
///             // ⇒ xTimeLimit := TRUE
///             // if the maximum operating time is reached
///             // ⇒ xTimeOut := TRUE
///             // if an error condition is reached
///             // ⇒ set iErrorID to a value other than 0 (Zero)
///             itfTimingController.ControllerCheckTiming(
///                 xTimeOut=>xTimeOut,
///                 xTimeLimit=>xTimeLimit
///             );
///         
///             xComplete := TRUE;
///             iErrorID := ERROR.NO_ERROR;
///     
///         UNTIL xComplete OR
///               xTimeOut OR xTimeLimit OR
///               iErrorID <> ERROR.NO_ERROR
///         END_REPEAT
///
/// .. note::
///
///    If this method will not provide any implementation, please remove it!
END_METHOD

METHOD ExitAction
VAR_INPUT
    xAfterCleanup : BOOL;
    xInCopyCode : BOOL;
END_VAR
{analysis -2} 
/// This method is intended for releasing external resources (like RTS handles).
/// Do not call other internal function block instances in the context of this method.
/// Call only external functions defined inside the RTS.
/// For cleaning up other resources then external ones, please use the ``CleanupAction``.
/// This method should be callable in the context of ``FB_EXIT`` for example
/// before downloading a new application or before reseting an application.
///
/// .. note::
///
///    If this method will not provide any implementation, please remove it!
END_METHOD

METHOD ResetAction
VAR_OUTPUT
    xComplete : BOOL := TRUE;
END_VAR
{analysis -2} 
/// The ``ResetAction`` is running until the output ``xComplete`` is ``TRUE``.
/// If ``xComplete`` is ``TRUE`` the state |STATE.DORMANT| is reached.
///
/// .. note::
///
///    If this method will not provide any implementation, please remove it!
END_METHOD

METHOD SampleAction
VAR_OUTPUT
 	iErrorID : INT := 0;
END_VAR
{analysis -2} 
/// After leaving the state |STATE.DORMANT| the ``SampleAction`` is running one time then the state |STATE.STARTING| is reached.
/// If there is a ``iErrorID`` ≠  0 (Zero) the state |STATE.CLEANING| is reached instead.
///
/// .. note::
///
///    If this method will not provide any implementation, please remove it!
END_METHOD

METHOD StartAction
VAR_OUTPUT
    xComplete : BOOL := TRUE;
	iErrorID : INT := 0;
END_VAR
{analysis -2} 
/// The ``StartAction`` is running until either the output ``xComplete`` is ``TRUE`` or ``iErrorID`` ≠ 0 (Zero).
/// If ``xComplete`` is ``TRUE`` the state |STATE.EXECUTING| is reached.
/// If there is a ``iErrorID`` ≠  0 (Zero) the state |STATE.CLEANING| is reached.
///
/// .. note::
///
///    To sample the inputs in the first invocation of a function block the method SampleAction is the solution of choice.
///    See: |ISampleActionProvider.SampleAction|
///
/// .. note::
///
///    If this method will not provide any implementation, please remove it!
END_METHOD

END_FUNCTION_BLOCK

// StringBuilder/Templates/Behaviour Model/ETrigTlTo_Temp
//{attribute 'hide_all_locals'}
//{attribute 'conditionalshow_all_locals' := 'SomeText'}
//{attribute 'conditionalshow_all_locals'}
//{attribute 'conditionalshow' := 'SomeText'}
//{attribute 'conditionalshow'}
//{attribute 'hide'}
FUNCTION_BLOCK ETrigTlTo_Temp EXTENDS CBML.ETrigTlTo
VAR_INPUT
	(* specific Inputs *)
END_VAR
VAR_OUTPUT
	eErrorID : ERROR;
	(* specific Outputs *)
END_VAR
VAR
	(* specific vars *)
END_VAR

SUPER^();
IF _Model.iErrorID = CBML.ERROR.TIME_OUT THEN
	eErrorID := ERROR.TIME_OUT;
ELSE
	eErrorID := _Model.iErrorID;
END_IF

METHOD CleanupAction
VAR_INPUT
    xAbortProposed : BOOL;
    iErrorIDProposed: INT;
END_VAR
VAR_OUTPUT
    xComplete : BOOL := TRUE;
    xAbort: BOOL := xAbortProposed;
 	iErrorID : INT := iErrorIDProposed;
END_VAR
{analysis -2} 
/// ``CleanupAction`` is running until one of the following events occurs:
/// When ``xComplete`` is ``TRUE`` the state |STATE.DONE| is reached.
/// When ``xAbort`` is ``TRUE`` the state |STATE.ABORTED| is reached.
/// When ``iErrorID`` ≠ 0 (Zero) the state |STATE.ERROR| is reached.
///
/// | After a *Ready Condition* as input (``iErrorIDProposed`` = 0 and ``xAbortProposed`` = ``FALSE``), only the output states
/// | `DONE` (``xComplete`` is ``TRUE``) or `ERROR` (``iErrorID`` ≠ 0) are possible.
///
/// | After a *Error Condition* as input (``iErrorIDProposed`` ≠ 0), only the output state
/// | `ERROR` (``iErrorID`` ≠ 0) is possible.
///
/// | After a *Abort Condition* as Input (``xAbortProposed`` = ``TRUE``), only the output states
/// | `ABORTED` (``xAbort`` is ``TRUE``) or `ERROR` (``iErrorID`` ≠ 0) are possible.
///
/// .. admonition:: Example
///
///     .. code-block:: codesys
///     
///         (* common cleanup -- first steps *) 
///         
///         IF xComplete THEN
///             IF xAbortProposed THEN
///                 (* abort condition -- abort specific cleanup *)
///                 xAbort := TRUE;
///                 xComplete := FALSE;
///             ELSIF iErrorIDProposed <> 0 THEN
///                 (* error condition -- error specific cleanup *)
///                 iErrorID := SEL(xComplete, 0, iErrorIDProposed);
///                 xComplete := FALSE;
///             ELSE
///                 (* ready condition -- done specific cleanup*)
///             END_IF
///         END_IF
///
///         (* common cleanup -- last steps *) 
///
/// .. note::
///
///    If this method will not provide any implementation, please remove it!
END_METHOD

METHOD CyclicAction
VAR_INPUT
    itfTimingController : CBML.ITimingController;
END_VAR
VAR_OUTPUT
    xComplete : BOOL := TRUE;
    iErrorID : INT := 0;
END_VAR
{analysis -2} 
/// The CyclicAction is running until either ``xComplete`` is ``TRUE`` or ``iErrorID`` ≠  0 (Zero).
/// If ``xComplete`` is ``TRUE`` or ``iErrorID`` ≠  0 (Zero) the state |STATE.CLEANING| is reached.
/// With ``itfTimingController`` ≠  0 (Zero) it is possible to check the current invocation time (see: |ITimingController.ControllerCheckTiming|).
/// Function blocks with a ``udiTimeLimit`` input variable (see: |IETrigTl|, |IETrigATl|, |IETrigTlTo|, |IETrigATlTo|, |ILConTl|, |ILConTlTo|, |ILConTlC|)
/// should be implement in such a way that the current invocation is exited when the consumed time for this invocation has exceeded the settings from udiTimeLimit.
///
/// .. admonition:: Example
///
///     .. code-block:: codesys
///     
///         REPEAT
///             // working to reach the ready condition
///             // ⇒ xComplete := TRUE
///             // if the maximum invocation time is reached
///             // ⇒ xTimeLimit := TRUE
///             // if the maximum operating time is reached
///             // ⇒ xTimeOut := TRUE
///             // if an error condition is reached
///             // ⇒ set iErrorID to a value other than 0 (Zero)
///             itfTimingController.ControllerCheckTiming(
///                 xTimeOut=>xTimeOut,
///                 xTimeLimit=>xTimeLimit
///             );
///         
///             xComplete := TRUE;
///             iErrorID := ERROR.NO_ERROR;
///     
///         UNTIL xComplete OR
///               xTimeOut OR xTimeLimit OR
///               iErrorID <> ERROR.NO_ERROR
///         END_REPEAT
///
/// .. note::
///
///    If this method will not provide any implementation, please remove it!
END_METHOD

METHOD ExitAction
VAR_INPUT
    xAfterCleanup : BOOL;
    xInCopyCode : BOOL;
END_VAR
{analysis -2} 
/// This method is intended for releasing external resources (like RTS handles).
/// Do not call other internal function block instances in the context of this method.
/// Call only external functions defined inside the RTS.
/// For cleaning up other resources then external ones, please use the ``CleanupAction``.
/// This method should be callable in the context of ``FB_EXIT`` for example
/// before downloading a new application or before reseting an application.
///
/// .. note::
///
///    If this method will not provide any implementation, please remove it!
END_METHOD

METHOD ResetAction
VAR_OUTPUT
    xComplete : BOOL := TRUE;
END_VAR
{analysis -2} 
/// The ``ResetAction`` is running until the output ``xComplete`` is ``TRUE``.
/// If ``xComplete`` is ``TRUE`` the state |STATE.DORMANT| is reached.
///
/// .. note::
///
///    If this method will not provide any implementation, please remove it!
END_METHOD

METHOD SampleAction
VAR_OUTPUT
 	iErrorID : INT := 0;
END_VAR
{analysis -2} 
/// After leaving the state |STATE.DORMANT| the ``SampleAction`` is running one time then the state |STATE.STARTING| is reached.
/// If there is a ``iErrorID`` ≠  0 (Zero) the state |STATE.CLEANING| is reached instead.
///
/// .. note::
///
///    If this method will not provide any implementation, please remove it!
END_METHOD

METHOD StartAction
VAR_OUTPUT
    xComplete : BOOL := TRUE;
	iErrorID : INT := 0;
END_VAR
{analysis -2} 
/// The ``StartAction`` is running until either the output ``xComplete`` is ``TRUE`` or ``iErrorID`` ≠ 0 (Zero).
/// If ``xComplete`` is ``TRUE`` the state |STATE.EXECUTING| is reached.
/// If there is a ``iErrorID`` ≠  0 (Zero) the state |STATE.CLEANING| is reached.
///
/// .. note::
///
///    To sample the inputs in the first invocation of a function block the method SampleAction is the solution of choice.
///    See: |ISampleActionProvider.SampleAction|
///
/// .. note::
///
///    If this method will not provide any implementation, please remove it!
END_METHOD

END_FUNCTION_BLOCK

// StringBuilder/Templates/Behaviour Model/ETrigTl_Temp
//{attribute 'hide_all_locals'}
//{attribute 'conditionalshow_all_locals' := 'SomeText'}
//{attribute 'conditionalshow_all_locals'}
//{attribute 'conditionalshow' := 'SomeText'}
//{attribute 'conditionalshow'}
//{attribute 'hide'}
FUNCTION_BLOCK ETrigTl_Temp EXTENDS CBML.ETrigTl
VAR_INPUT
	(* specific Inputs *)
END_VAR
VAR_OUTPUT
	eErrorID : ERROR;
	(* specific Outputs *)
END_VAR
VAR
	(* specific vars *)
END_VAR

SUPER^();
eErrorID := _Model.iErrorID;

METHOD CleanupAction
VAR_INPUT
    xAbortProposed : BOOL;
    iErrorIDProposed: INT;
END_VAR
VAR_OUTPUT
    xComplete : BOOL := TRUE;
    xAbort: BOOL := xAbortProposed;
 	iErrorID : INT := iErrorIDProposed;
END_VAR
{analysis -2} 
/// ``CleanupAction`` is running until one of the following events occurs:
/// When ``xComplete`` is ``TRUE`` the state |STATE.DONE| is reached.
/// When ``xAbort`` is ``TRUE`` the state |STATE.ABORTED| is reached.
/// When ``iErrorID`` ≠ 0 (Zero) the state |STATE.ERROR| is reached.
///
/// | After a *Ready Condition* as input (``iErrorIDProposed`` = 0 and ``xAbortProposed`` = ``FALSE``), only the output states
/// | `DONE` (``xComplete`` is ``TRUE``) or `ERROR` (``iErrorID`` ≠ 0) are possible.
///
/// | After a *Error Condition* as input (``iErrorIDProposed`` ≠ 0), only the output state
/// | `ERROR` (``iErrorID`` ≠ 0) is possible.
///
/// | After a *Abort Condition* as Input (``xAbortProposed`` = ``TRUE``), only the output states
/// | `ABORTED` (``xAbort`` is ``TRUE``) or `ERROR` (``iErrorID`` ≠ 0) are possible.
///
/// .. admonition:: Example
///
///     .. code-block:: codesys
///     
///         (* common cleanup -- first steps *) 
///         
///         IF xComplete THEN
///             IF xAbortProposed THEN
///                 (* abort condition -- abort specific cleanup *)
///                 xAbort := TRUE;
///                 xComplete := FALSE;
///             ELSIF iErrorIDProposed <> 0 THEN
///                 (* error condition -- error specific cleanup *)
///                 iErrorID := SEL(xComplete, 0, iErrorIDProposed);
///                 xComplete := FALSE;
///             ELSE
///                 (* ready condition -- done specific cleanup*)
///             END_IF
///         END_IF
///
///         (* common cleanup -- last steps *) 
///
/// .. note::
///
///    If this method will not provide any implementation, please remove it!
END_METHOD

METHOD CyclicAction
VAR_INPUT
    itfTimingController : CBML.ITimingController;
END_VAR
VAR_OUTPUT
    xComplete : BOOL := TRUE;
    iErrorID : INT := 0;
END_VAR
{analysis -2} 
/// The CyclicAction is running until either ``xComplete`` is ``TRUE`` or ``iErrorID`` ≠  0 (Zero).
/// If ``xComplete`` is ``TRUE`` or ``iErrorID`` ≠  0 (Zero) the state |STATE.CLEANING| is reached.
/// With ``itfTimingController`` ≠  0 (Zero) it is possible to check the current invocation time (see: |ITimingController.ControllerCheckTiming|).
/// Function blocks with a ``udiTimeLimit`` input variable (see: |IETrigTl|, |IETrigATl|, |IETrigTlTo|, |IETrigATlTo|, |ILConTl|, |ILConTlTo|, |ILConTlC|)
/// should be implement in such a way that the current invocation is exited when the consumed time for this invocation has exceeded the settings from udiTimeLimit.
///
/// .. admonition:: Example
///
///     .. code-block:: codesys
///     
///         REPEAT
///             // working to reach the ready condition
///             // ⇒ xComplete := TRUE
///             // if the maximum invocation time is reached
///             // ⇒ xTimeLimit := TRUE
///             // if the maximum operating time is reached
///             // ⇒ xTimeOut := TRUE
///             // if an error condition is reached
///             // ⇒ set iErrorID to a value other than 0 (Zero)
///             itfTimingController.ControllerCheckTiming(
///                 xTimeOut=>xTimeOut,
///                 xTimeLimit=>xTimeLimit
///             );
///         
///             xComplete := TRUE;
///             iErrorID := ERROR.NO_ERROR;
///     
///         UNTIL xComplete OR
///               xTimeOut OR xTimeLimit OR
///               iErrorID <> ERROR.NO_ERROR
///         END_REPEAT
///
/// .. note::
///
///    If this method will not provide any implementation, please remove it!
END_METHOD

METHOD ExitAction
VAR_INPUT
    xAfterCleanup : BOOL;
    xInCopyCode : BOOL;
END_VAR
{analysis -2} 
/// This method is intended for releasing external resources (like RTS handles).
/// Do not call other internal function block instances in the context of this method.
/// Call only external functions defined inside the RTS.
/// For cleaning up other resources then external ones, please use the ``CleanupAction``.
/// This method should be callable in the context of ``FB_EXIT`` for example
/// before downloading a new application or before reseting an application.
///
/// .. note::
///
///    If this method will not provide any implementation, please remove it!
END_METHOD

METHOD ResetAction
VAR_OUTPUT
    xComplete : BOOL := TRUE;
END_VAR
{analysis -2} 
/// The ``ResetAction`` is running until the output ``xComplete`` is ``TRUE``.
/// If ``xComplete`` is ``TRUE`` the state |STATE.DORMANT| is reached.
///
/// .. note::
///
///    If this method will not provide any implementation, please remove it!
END_METHOD

METHOD SampleAction
VAR_OUTPUT
 	iErrorID : INT := 0;
END_VAR
{analysis -2} 
/// After leaving the state |STATE.DORMANT| the ``SampleAction`` is running one time then the state |STATE.STARTING| is reached.
/// If there is a ``iErrorID`` ≠  0 (Zero) the state |STATE.CLEANING| is reached instead.
///
/// .. note::
///
///    If this method will not provide any implementation, please remove it!
END_METHOD

METHOD StartAction
VAR_OUTPUT
    xComplete : BOOL := TRUE;
	iErrorID : INT := 0;
END_VAR
{analysis -2} 
/// The ``StartAction`` is running until either the output ``xComplete`` is ``TRUE`` or ``iErrorID`` ≠ 0 (Zero).
/// If ``xComplete`` is ``TRUE`` the state |STATE.EXECUTING| is reached.
/// If there is a ``iErrorID`` ≠  0 (Zero) the state |STATE.CLEANING| is reached.
///
/// .. note::
///
///    To sample the inputs in the first invocation of a function block the method SampleAction is the solution of choice.
///    See: |ISampleActionProvider.SampleAction|
///
/// .. note::
///
///    If this method will not provide any implementation, please remove it!
END_METHOD

END_FUNCTION_BLOCK

// StringBuilder/Templates/Behaviour Model/ETrigTo_Temp
//{attribute 'hide_all_locals'}
//{attribute 'conditionalshow_all_locals' := 'SomeText'}
//{attribute 'conditionalshow_all_locals'}
//{attribute 'conditionalshow' := 'SomeText'}
//{attribute 'conditionalshow'}
//{attribute 'hide'}
FUNCTION_BLOCK ETrigTo_Temp EXTENDS CBML.ETrigTo
VAR_INPUT
	(* specific Inputs *)
END_VAR
VAR_OUTPUT
	eErrorID : ERROR;
	(* specific Outputs *)
END_VAR
VAR
	(* specific vars *)
END_VAR

SUPER^();
IF _Model.iErrorID = CBML.ERROR.TIME_OUT THEN
	eErrorID := ERROR.TIME_OUT;
ELSE
	eErrorID := _Model.iErrorID;
END_IF

METHOD CleanupAction
VAR_INPUT
    xAbortProposed : BOOL;
    iErrorIDProposed: INT;
END_VAR
VAR_OUTPUT
    xComplete : BOOL := TRUE;
    xAbort: BOOL := xAbortProposed;
 	iErrorID : INT := iErrorIDProposed;
END_VAR
{analysis -2} 
/// ``CleanupAction`` is running until one of the following events occurs:
/// When ``xComplete`` is ``TRUE`` the state |STATE.DONE| is reached.
/// When ``xAbort`` is ``TRUE`` the state |STATE.ABORTED| is reached.
/// When ``iErrorID`` ≠ 0 (Zero) the state |STATE.ERROR| is reached.
///
/// | After a *Ready Condition* as input (``iErrorIDProposed`` = 0 and ``xAbortProposed`` = ``FALSE``), only the output states
/// | `DONE` (``xComplete`` is ``TRUE``) or `ERROR` (``iErrorID`` ≠ 0) are possible.
///
/// | After a *Error Condition* as input (``iErrorIDProposed`` ≠ 0), only the output state
/// | `ERROR` (``iErrorID`` ≠ 0) is possible.
///
/// | After a *Abort Condition* as Input (``xAbortProposed`` = ``TRUE``), only the output states
/// | `ABORTED` (``xAbort`` is ``TRUE``) or `ERROR` (``iErrorID`` ≠ 0) are possible.
///
/// .. admonition:: Example
///
///     .. code-block:: codesys
///     
///         (* common cleanup -- first steps *) 
///         
///         IF xComplete THEN
///             IF xAbortProposed THEN
///                 (* abort condition -- abort specific cleanup *)
///                 xAbort := TRUE;
///                 xComplete := FALSE;
///             ELSIF iErrorIDProposed <> 0 THEN
///                 (* error condition -- error specific cleanup *)
///                 iErrorID := SEL(xComplete, 0, iErrorIDProposed);
///                 xComplete := FALSE;
///             ELSE
///                 (* ready condition -- done specific cleanup*)
///             END_IF
///         END_IF
///
///         (* common cleanup -- last steps *) 
///
/// .. note::
///
///    If this method will not provide any implementation, please remove it!
END_METHOD

METHOD CyclicAction
VAR_INPUT
    itfTimingController : CBML.ITimingController;
END_VAR
VAR_OUTPUT
    xComplete : BOOL := TRUE;
    iErrorID : INT := 0;
END_VAR
{analysis -2} 
/// The CyclicAction is running until either ``xComplete`` is ``TRUE`` or ``iErrorID`` ≠  0 (Zero).
/// If ``xComplete`` is ``TRUE`` or ``iErrorID`` ≠  0 (Zero) the state |STATE.CLEANING| is reached.
/// With ``itfTimingController`` ≠  0 (Zero) it is possible to check the current invocation time (see: |ITimingController.ControllerCheckTiming|).
/// Function blocks with a ``udiTimeLimit`` input variable (see: |IETrigTl|, |IETrigATl|, |IETrigTlTo|, |IETrigATlTo|, |ILConTl|, |ILConTlTo|, |ILConTlC|)
/// should be implement in such a way that the current invocation is exited when the consumed time for this invocation has exceeded the settings from udiTimeLimit.
///
/// .. admonition:: Example
///
///     .. code-block:: codesys
///     
///         REPEAT
///             // working to reach the ready condition
///             // ⇒ xComplete := TRUE
///             // if the maximum invocation time is reached
///             // ⇒ xTimeLimit := TRUE
///             // if the maximum operating time is reached
///             // ⇒ xTimeOut := TRUE
///             // if an error condition is reached
///             // ⇒ set iErrorID to a value other than 0 (Zero)
///             itfTimingController.ControllerCheckTiming(
///                 xTimeOut=>xTimeOut,
///                 xTimeLimit=>xTimeLimit
///             );
///         
///             xComplete := TRUE;
///             iErrorID := ERROR.NO_ERROR;
///     
///         UNTIL xComplete OR
///               xTimeOut OR xTimeLimit OR
///               iErrorID <> ERROR.NO_ERROR
///         END_REPEAT
///
/// .. note::
///
///    If this method will not provide any implementation, please remove it!
END_METHOD

METHOD ExitAction
VAR_INPUT
    xAfterCleanup : BOOL;
    xInCopyCode : BOOL;
END_VAR
{analysis -2} 
/// This method is intended for releasing external resources (like RTS handles).
/// Do not call other internal function block instances in the context of this method.
/// Call only external functions defined inside the RTS.
/// For cleaning up other resources then external ones, please use the ``CleanupAction``.
/// This method should be callable in the context of ``FB_EXIT`` for example
/// before downloading a new application or before reseting an application.
///
/// .. note::
///
///    If this method will not provide any implementation, please remove it!
END_METHOD

METHOD ResetAction
VAR_OUTPUT
    xComplete : BOOL := TRUE;
END_VAR
{analysis -2} 
/// The ``ResetAction`` is running until the output ``xComplete`` is ``TRUE``.
/// If ``xComplete`` is ``TRUE`` the state |STATE.DORMANT| is reached.
///
/// .. note::
///
///    If this method will not provide any implementation, please remove it!
END_METHOD

METHOD SampleAction
VAR_OUTPUT
 	iErrorID : INT := 0;
END_VAR
{analysis -2} 
/// After leaving the state |STATE.DORMANT| the ``SampleAction`` is running one time then the state |STATE.STARTING| is reached.
/// If there is a ``iErrorID`` ≠  0 (Zero) the state |STATE.CLEANING| is reached instead.
///
/// .. note::
///
///    If this method will not provide any implementation, please remove it!
END_METHOD

METHOD StartAction
VAR_OUTPUT
    xComplete : BOOL := TRUE;
	iErrorID : INT := 0;
END_VAR
{analysis -2} 
/// The ``StartAction`` is running until either the output ``xComplete`` is ``TRUE`` or ``iErrorID`` ≠ 0 (Zero).
/// If ``xComplete`` is ``TRUE`` the state |STATE.EXECUTING| is reached.
/// If there is a ``iErrorID`` ≠  0 (Zero) the state |STATE.CLEANING| is reached.
///
/// .. note::
///
///    To sample the inputs in the first invocation of a function block the method SampleAction is the solution of choice.
///    See: |ISampleActionProvider.SampleAction|
///
/// .. note::
///
///    If this method will not provide any implementation, please remove it!
END_METHOD

END_FUNCTION_BLOCK

// StringBuilder/Templates/Behaviour Model/ETrig_Temp
//{attribute 'hide_all_locals'}
//{attribute 'conditionalshow_all_locals' := 'SomeText'}
//{attribute 'conditionalshow_all_locals'}
//{attribute 'conditionalshow' := 'SomeText'}
//{attribute 'conditionalshow'}
//{attribute 'hide'}
FUNCTION_BLOCK ETrig_Temp EXTENDS CBML.ETrig
VAR_INPUT
	(* specific Inputs *)
END_VAR
VAR_OUTPUT
	eErrorID : ERROR;
	(* specific Outputs *)
END_VAR
VAR
	(* specific vars *)
END_VAR

SUPER^();
eErrorID := _Model.iErrorID;

METHOD CleanupAction
VAR_INPUT
    xAbortProposed : BOOL;
    iErrorIDProposed: INT;
END_VAR
VAR_OUTPUT
    xComplete : BOOL := TRUE;
    xAbort: BOOL := xAbortProposed;
 	iErrorID : INT := iErrorIDProposed;
END_VAR
{analysis -2} 
/// ``CleanupAction`` is running until one of the following events occurs:
/// When ``xComplete`` is ``TRUE`` the state |STATE.DONE| is reached.
/// When ``xAbort`` is ``TRUE`` the state |STATE.ABORTED| is reached.
/// When ``iErrorID`` ≠ 0 (Zero) the state |STATE.ERROR| is reached.
///
/// | After a *Ready Condition* as input (``iErrorIDProposed`` = 0 and ``xAbortProposed`` = ``FALSE``), only the output states
/// | `DONE` (``xComplete`` is ``TRUE``) or `ERROR` (``iErrorID`` ≠ 0) are possible.
///
/// | After a *Error Condition* as input (``iErrorIDProposed`` ≠ 0), only the output state
/// | `ERROR` (``iErrorID`` ≠ 0) is possible.
///
/// | After a *Abort Condition* as Input (``xAbortProposed`` = ``TRUE``), only the output states
/// | `ABORTED` (``xAbort`` is ``TRUE``) or `ERROR` (``iErrorID`` ≠ 0) are possible.
///
/// .. admonition:: Example
///
///     .. code-block:: codesys
///     
///         (* common cleanup -- first steps *) 
///         
///         IF xComplete THEN
///             IF xAbortProposed THEN
///                 (* abort condition -- abort specific cleanup *)
///                 xAbort := TRUE;
///                 xComplete := FALSE;
///             ELSIF iErrorIDProposed <> 0 THEN
///                 (* error condition -- error specific cleanup *)
///                 iErrorID := SEL(xComplete, 0, iErrorIDProposed);
///                 xComplete := FALSE;
///             ELSE
///                 (* ready condition -- done specific cleanup*)
///             END_IF
///         END_IF
///
///         (* common cleanup -- last steps *) 
///
/// .. note::
///
///    If this method will not provide any implementation, please remove it!
END_METHOD

METHOD CyclicAction
VAR_INPUT
    itfTimingController : CBML.ITimingController;
END_VAR
VAR_OUTPUT
    xComplete : BOOL := TRUE;
    iErrorID : INT := 0;
END_VAR
{analysis -2} 
/// The CyclicAction is running until either ``xComplete`` is ``TRUE`` or ``iErrorID`` ≠  0 (Zero).
/// If ``xComplete`` is ``TRUE`` or ``iErrorID`` ≠  0 (Zero) the state |STATE.CLEANING| is reached.
/// With ``itfTimingController`` ≠  0 (Zero) it is possible to check the current invocation time (see: |ITimingController.ControllerCheckTiming|).
/// Function blocks with a ``udiTimeLimit`` input variable (see: |IETrigTl|, |IETrigATl|, |IETrigTlTo|, |IETrigATlTo|, |ILConTl|, |ILConTlTo|, |ILConTlC|)
/// should be implement in such a way that the current invocation is exited when the consumed time for this invocation has exceeded the settings from udiTimeLimit.
///
/// .. admonition:: Example
///
///     .. code-block:: codesys
///     
///         REPEAT
///             // working to reach the ready condition
///             // ⇒ xComplete := TRUE
///             // if the maximum invocation time is reached
///             // ⇒ xTimeLimit := TRUE
///             // if the maximum operating time is reached
///             // ⇒ xTimeOut := TRUE
///             // if an error condition is reached
///             // ⇒ set iErrorID to a value other than 0 (Zero)
///             itfTimingController.ControllerCheckTiming(
///                 xTimeOut=>xTimeOut,
///                 xTimeLimit=>xTimeLimit
///             );
///         
///             xComplete := TRUE;
///             iErrorID := ERROR.NO_ERROR;
///     
///         UNTIL xComplete OR
///               xTimeOut OR xTimeLimit OR
///               iErrorID <> ERROR.NO_ERROR
///         END_REPEAT
///
/// .. note::
///
///    If this method will not provide any implementation, please remove it!
END_METHOD

METHOD ExitAction
VAR_INPUT
    xAfterCleanup : BOOL;
    xInCopyCode : BOOL;
END_VAR
{analysis -2} 
/// This method is intended for releasing external resources (like RTS handles).
/// Do not call other internal function block instances in the context of this method.
/// Call only external functions defined inside the RTS.
/// For cleaning up other resources then external ones, please use the ``CleanupAction``.
/// This method should be callable in the context of ``FB_EXIT`` for example
/// before downloading a new application or before reseting an application.
///
/// .. note::
///
///    If this method will not provide any implementation, please remove it!
END_METHOD

METHOD ResetAction
VAR_OUTPUT
    xComplete : BOOL := TRUE;
END_VAR
{analysis -2} 
/// The ``ResetAction`` is running until the output ``xComplete`` is ``TRUE``.
/// If ``xComplete`` is ``TRUE`` the state |STATE.DORMANT| is reached.
///
/// .. note::
///
///    If this method will not provide any implementation, please remove it!
END_METHOD

METHOD SampleAction
VAR_OUTPUT
 	iErrorID : INT := 0;
END_VAR
{analysis -2} 
/// After leaving the state |STATE.DORMANT| the ``SampleAction`` is running one time then the state |STATE.STARTING| is reached.
/// If there is a ``iErrorID`` ≠  0 (Zero) the state |STATE.CLEANING| is reached instead.
///
/// .. note::
///
///    If this method will not provide any implementation, please remove it!
END_METHOD

METHOD StartAction
VAR_OUTPUT
    xComplete : BOOL := TRUE;
	iErrorID : INT := 0;
END_VAR
{analysis -2} 
/// The ``StartAction`` is running until either the output ``xComplete`` is ``TRUE`` or ``iErrorID`` ≠ 0 (Zero).
/// If ``xComplete`` is ``TRUE`` the state |STATE.EXECUTING| is reached.
/// If there is a ``iErrorID`` ≠  0 (Zero) the state |STATE.CLEANING| is reached.
///
/// .. note::
///
///    To sample the inputs in the first invocation of a function block the method SampleAction is the solution of choice.
///    See: |ISampleActionProvider.SampleAction|
///
/// .. note::
///
///    If this method will not provide any implementation, please remove it!
END_METHOD

END_FUNCTION_BLOCK

// StringBuilder/Templates/Behaviour Model/LConC_Temp
//{attribute 'hide_all_locals'}
//{attribute 'conditionalshow_all_locals' := 'SomeText'}
//{attribute 'conditionalshow_all_locals'}
//{attribute 'conditionalshow' := 'SomeText'}
//{attribute 'conditionalshow'}
//{attribute 'hide'}
FUNCTION_BLOCK LConC_Temp EXTENDS CBML.LConC
VAR_INPUT
	(* specific Inputs *)
END_VAR
VAR_OUTPUT
	eErrorID : ERROR;
	(* specific Outputs *)
END_VAR
VAR
	(* specific vars *)
END_VAR

SUPER^();
eErrorID := _Model.iErrorID;

METHOD CleanupAction
VAR_INPUT
    xAbortProposed : BOOL;
    iErrorIDProposed: INT;
END_VAR
VAR_OUTPUT
    xComplete : BOOL := TRUE;
    xAbort: BOOL := xAbortProposed;
 	iErrorID : INT := iErrorIDProposed;
END_VAR
{analysis -2} 
/// ``CleanupAction`` is running until one of the following events occurs:
/// When ``xComplete`` is ``TRUE`` the state |STATE.DONE| is reached.
/// When ``xAbort`` is ``TRUE`` the state |STATE.ABORTED| is reached.
/// When ``iErrorID`` ≠ 0 (Zero) the state |STATE.ERROR| is reached.
///
/// | After a *Ready Condition* as input (``iErrorIDProposed`` = 0 and ``xAbortProposed`` = ``FALSE``), only the output states
/// | `DONE` (``xComplete`` is ``TRUE``) or `ERROR` (``iErrorID`` ≠ 0) are possible.
///
/// | After a *Error Condition* as input (``iErrorIDProposed`` ≠ 0), only the output state
/// | `ERROR` (``iErrorID`` ≠ 0) is possible.
///
/// | After a *Abort Condition* as Input (``xAbortProposed`` = ``TRUE``), only the output states
/// | `ABORTED` (``xAbort`` is ``TRUE``) or `ERROR` (``iErrorID`` ≠ 0) are possible.
///
/// .. admonition:: Example
///
///     .. code-block:: codesys
///     
///         (* common cleanup -- first steps *) 
///         
///         IF xComplete THEN
///             IF xAbortProposed THEN
///                 (* abort condition -- abort specific cleanup *)
///                 xAbort := TRUE;
///                 xComplete := FALSE;
///             ELSIF iErrorIDProposed <> 0 THEN
///                 (* error condition -- error specific cleanup *)
///                 iErrorID := SEL(xComplete, 0, iErrorIDProposed);
///                 xComplete := FALSE;
///             ELSE
///                 (* ready condition -- done specific cleanup*)
///             END_IF
///         END_IF
///
///         (* common cleanup -- last steps *) 
///
/// .. note::
///
///    If this method will not provide any implementation, please remove it!
END_METHOD

METHOD CyclicAction
VAR_INPUT
    itfTimingController : CBML.ITimingController;
END_VAR
VAR_OUTPUT
    xComplete : BOOL := TRUE;
    iErrorID : INT := 0;
END_VAR
{analysis -2} 
/// The CyclicAction is running until either ``xComplete`` is ``TRUE`` or ``iErrorID`` ≠  0 (Zero).
/// If ``xComplete`` is ``TRUE`` or ``iErrorID`` ≠  0 (Zero) the state |STATE.CLEANING| is reached.
/// With ``itfTimingController`` ≠  0 (Zero) it is possible to check the current invocation time (see: |ITimingController.ControllerCheckTiming|).
/// Function blocks with a ``udiTimeLimit`` input variable (see: |IETrigTl|, |IETrigATl|, |IETrigTlTo|, |IETrigATlTo|, |ILConTl|, |ILConTlTo|, |ILConTlC|)
/// should be implement in such a way that the current invocation is exited when the consumed time for this invocation has exceeded the settings from udiTimeLimit.
///
/// .. admonition:: Example
///
///     .. code-block:: codesys
///     
///         REPEAT
///             // working to reach the ready condition
///             // ⇒ xComplete := TRUE
///             // if the maximum invocation time is reached
///             // ⇒ xTimeLimit := TRUE
///             // if the maximum operating time is reached
///             // ⇒ xTimeOut := TRUE
///             // if an error condition is reached
///             // ⇒ set iErrorID to a value other than 0 (Zero)
///             itfTimingController.ControllerCheckTiming(
///                 xTimeOut=>xTimeOut,
///                 xTimeLimit=>xTimeLimit
///             );
///         
///             xComplete := TRUE;
///             iErrorID := ERROR.NO_ERROR;
///     
///         UNTIL xComplete OR
///               xTimeOut OR xTimeLimit OR
///               iErrorID <> ERROR.NO_ERROR
///         END_REPEAT
///
/// .. note::
///
///    If this method will not provide any implementation, please remove it!
END_METHOD

METHOD ExitAction
VAR_INPUT
    xAfterCleanup : BOOL;
    xInCopyCode : BOOL;
END_VAR
{analysis -2} 
/// This method is intended for releasing external resources (like RTS handles).
/// Do not call other internal function block instances in the context of this method.
/// Call only external functions defined inside the RTS.
/// For cleaning up other resources then external ones, please use the ``CleanupAction``.
/// This method should be callable in the context of ``FB_EXIT`` for example
/// before downloading a new application or before reseting an application.
///
/// .. note::
///
///    If this method will not provide any implementation, please remove it!
END_METHOD

METHOD ResetAction
VAR_OUTPUT
    xComplete : BOOL := TRUE;
END_VAR
{analysis -2} 
/// The ``ResetAction`` is running until the output ``xComplete`` is ``TRUE``.
/// If ``xComplete`` is ``TRUE`` the state |STATE.DORMANT| is reached.
///
/// .. note::
///
///    If this method will not provide any implementation, please remove it!
END_METHOD

METHOD StartAction
VAR_OUTPUT
    xComplete : BOOL := TRUE;
	iErrorID : INT := 0;
END_VAR
{analysis -2} 
/// The ``StartAction`` is running until either the output ``xComplete`` is ``TRUE`` or ``iErrorID`` ≠ 0 (Zero).
/// If ``xComplete`` is ``TRUE`` the state |STATE.EXECUTING| is reached.
/// If there is a ``iErrorID`` ≠  0 (Zero) the state |STATE.CLEANING| is reached.
///
/// .. note::
///
///    To sample the inputs in the first invocation of a function block the method SampleAction is the solution of choice.
///    See: |ISampleActionProvider.SampleAction|
///
/// .. note::
///
///    If this method will not provide any implementation, please remove it!
END_METHOD

END_FUNCTION_BLOCK

// StringBuilder/Templates/Behaviour Model/LConTlC_Temp
//{attribute 'hide_all_locals'}
//{attribute 'conditionalshow_all_locals' := 'SomeText'}
//{attribute 'conditionalshow_all_locals'}
//{attribute 'conditionalshow' := 'SomeText'}
//{attribute 'conditionalshow'}
//{attribute 'hide'}
FUNCTION_BLOCK LConTlC_Temp EXTENDS CBML.LConTlC
VAR_INPUT
	(* specific Inputs *)
END_VAR
VAR_OUTPUT
	eErrorID : ERROR;
	(* specific Outputs *)
END_VAR
VAR
	(* specific vars *)
END_VAR

SUPER^();
eErrorID := _Model.iErrorID;

METHOD CleanupAction
VAR_INPUT
    xAbortProposed : BOOL;
    iErrorIDProposed: INT;
END_VAR
VAR_OUTPUT
    xComplete : BOOL := TRUE;
    xAbort: BOOL := xAbortProposed;
 	iErrorID : INT := iErrorIDProposed;
END_VAR
{analysis -2} 
/// ``CleanupAction`` is running until one of the following events occurs:
/// When ``xComplete`` is ``TRUE`` the state |STATE.DONE| is reached.
/// When ``xAbort`` is ``TRUE`` the state |STATE.ABORTED| is reached.
/// When ``iErrorID`` ≠ 0 (Zero) the state |STATE.ERROR| is reached.
///
/// | After a *Ready Condition* as input (``iErrorIDProposed`` = 0 and ``xAbortProposed`` = ``FALSE``), only the output states
/// | `DONE` (``xComplete`` is ``TRUE``) or `ERROR` (``iErrorID`` ≠ 0) are possible.
///
/// | After a *Error Condition* as input (``iErrorIDProposed`` ≠ 0), only the output state
/// | `ERROR` (``iErrorID`` ≠ 0) is possible.
///
/// | After a *Abort Condition* as Input (``xAbortProposed`` = ``TRUE``), only the output states
/// | `ABORTED` (``xAbort`` is ``TRUE``) or `ERROR` (``iErrorID`` ≠ 0) are possible.
///
/// .. admonition:: Example
///
///     .. code-block:: codesys
///     
///         (* common cleanup -- first steps *) 
///         
///         IF xComplete THEN
///             IF xAbortProposed THEN
///                 (* abort condition -- abort specific cleanup *)
///                 xAbort := TRUE;
///                 xComplete := FALSE;
///             ELSIF iErrorIDProposed <> 0 THEN
///                 (* error condition -- error specific cleanup *)
///                 iErrorID := SEL(xComplete, 0, iErrorIDProposed);
///                 xComplete := FALSE;
///             ELSE
///                 (* ready condition -- done specific cleanup*)
///             END_IF
///         END_IF
///
///         (* common cleanup -- last steps *) 
///
/// .. note::
///
///    If this method will not provide any implementation, please remove it!
END_METHOD

METHOD CyclicAction
VAR_INPUT
    itfTimingController : CBML.ITimingController;
END_VAR
VAR_OUTPUT
    xComplete : BOOL := TRUE;
    iErrorID : INT := 0;
END_VAR
{analysis -2} 
/// The CyclicAction is running until either ``xComplete`` is ``TRUE`` or ``iErrorID`` ≠  0 (Zero).
/// If ``xComplete`` is ``TRUE`` or ``iErrorID`` ≠  0 (Zero) the state |STATE.CLEANING| is reached.
/// With ``itfTimingController`` ≠  0 (Zero) it is possible to check the current invocation time (see: |ITimingController.ControllerCheckTiming|).
/// Function blocks with a ``udiTimeLimit`` input variable (see: |IETrigTl|, |IETrigATl|, |IETrigTlTo|, |IETrigATlTo|, |ILConTl|, |ILConTlTo|, |ILConTlC|)
/// should be implement in such a way that the current invocation is exited when the consumed time for this invocation has exceeded the settings from udiTimeLimit.
///
/// .. admonition:: Example
///
///     .. code-block:: codesys
///     
///         REPEAT
///             // working to reach the ready condition
///             // ⇒ xComplete := TRUE
///             // if the maximum invocation time is reached
///             // ⇒ xTimeLimit := TRUE
///             // if the maximum operating time is reached
///             // ⇒ xTimeOut := TRUE
///             // if an error condition is reached
///             // ⇒ set iErrorID to a value other than 0 (Zero)
///             itfTimingController.ControllerCheckTiming(
///                 xTimeOut=>xTimeOut,
///                 xTimeLimit=>xTimeLimit
///             );
///         
///             xComplete := TRUE;
///             iErrorID := ERROR.NO_ERROR;
///     
///         UNTIL xComplete OR
///               xTimeOut OR xTimeLimit OR
///               iErrorID <> ERROR.NO_ERROR
///         END_REPEAT
///
/// .. note::
///
///    If this method will not provide any implementation, please remove it!
END_METHOD

METHOD ExitAction
VAR_INPUT
    xAfterCleanup : BOOL;
    xInCopyCode : BOOL;
END_VAR
{analysis -2} 
/// This method is intended for releasing external resources (like RTS handles).
/// Do not call other internal function block instances in the context of this method.
/// Call only external functions defined inside the RTS.
/// For cleaning up other resources then external ones, please use the ``CleanupAction``.
/// This method should be callable in the context of ``FB_EXIT`` for example
/// before downloading a new application or before reseting an application.
///
/// .. note::
///
///    If this method will not provide any implementation, please remove it!
END_METHOD

METHOD ResetAction
VAR_OUTPUT
    xComplete : BOOL := TRUE;
END_VAR
{analysis -2} 
/// The ``ResetAction`` is running until the output ``xComplete`` is ``TRUE``.
/// If ``xComplete`` is ``TRUE`` the state |STATE.DORMANT| is reached.
///
/// .. note::
///
///    If this method will not provide any implementation, please remove it!
END_METHOD

METHOD StartAction
VAR_OUTPUT
    xComplete : BOOL := TRUE;
	iErrorID : INT := 0;
END_VAR
{analysis -2} 
/// The ``StartAction`` is running until either the output ``xComplete`` is ``TRUE`` or ``iErrorID`` ≠ 0 (Zero).
/// If ``xComplete`` is ``TRUE`` the state |STATE.EXECUTING| is reached.
/// If there is a ``iErrorID`` ≠  0 (Zero) the state |STATE.CLEANING| is reached.
///
/// .. note::
///
///    To sample the inputs in the first invocation of a function block the method SampleAction is the solution of choice.
///    See: |ISampleActionProvider.SampleAction|
///
/// .. note::
///
///    If this method will not provide any implementation, please remove it!
END_METHOD

END_FUNCTION_BLOCK

// StringBuilder/Templates/Behaviour Model/LConTlTo_Temp
//{attribute 'hide_all_locals'}
//{attribute 'conditionalshow_all_locals' := 'SomeText'}
//{attribute 'conditionalshow_all_locals'}
//{attribute 'conditionalshow' := 'SomeText'}
//{attribute 'conditionalshow'}
//{attribute 'hide'}
FUNCTION_BLOCK LConTlTo_Temp EXTENDS CBML.LConTlTo
VAR_INPUT
	(* specific Inputs *)
END_VAR
VAR_OUTPUT
	eErrorID : ERROR;
	(* specific Outputs *)
END_VAR
VAR
	(* specific vars *)
END_VAR

SUPER^();
IF _Model.iErrorID = CBML.ERROR.TIME_OUT THEN
	eErrorID := ERROR.TIME_OUT;
ELSE
	eErrorID := _Model.iErrorID;
END_IF

METHOD CleanupAction
VAR_INPUT
    xAbortProposed : BOOL;
    iErrorIDProposed: INT;
END_VAR
VAR_OUTPUT
    xComplete : BOOL := TRUE;
    xAbort: BOOL := xAbortProposed;
 	iErrorID : INT := iErrorIDProposed;
END_VAR
{analysis -2} 
/// ``CleanupAction`` is running until one of the following events occurs:
/// When ``xComplete`` is ``TRUE`` the state |STATE.DONE| is reached.
/// When ``xAbort`` is ``TRUE`` the state |STATE.ABORTED| is reached.
/// When ``iErrorID`` ≠ 0 (Zero) the state |STATE.ERROR| is reached.
///
/// | After a *Ready Condition* as input (``iErrorIDProposed`` = 0 and ``xAbortProposed`` = ``FALSE``), only the output states
/// | `DONE` (``xComplete`` is ``TRUE``) or `ERROR` (``iErrorID`` ≠ 0) are possible.
///
/// | After a *Error Condition* as input (``iErrorIDProposed`` ≠ 0), only the output state
/// | `ERROR` (``iErrorID`` ≠ 0) is possible.
///
/// | After a *Abort Condition* as Input (``xAbortProposed`` = ``TRUE``), only the output states
/// | `ABORTED` (``xAbort`` is ``TRUE``) or `ERROR` (``iErrorID`` ≠ 0) are possible.
///
/// .. admonition:: Example
///
///     .. code-block:: codesys
///     
///         (* common cleanup -- first steps *) 
///         
///         IF xComplete THEN
///             IF xAbortProposed THEN
///                 (* abort condition -- abort specific cleanup *)
///                 xAbort := TRUE;
///                 xComplete := FALSE;
///             ELSIF iErrorIDProposed <> 0 THEN
///                 (* error condition -- error specific cleanup *)
///                 iErrorID := SEL(xComplete, 0, iErrorIDProposed);
///                 xComplete := FALSE;
///             ELSE
///                 (* ready condition -- done specific cleanup*)
///             END_IF
///         END_IF
///
///         (* common cleanup -- last steps *) 
///
/// .. note::
///
///    If this method will not provide any implementation, please remove it!
END_METHOD

